Universal Robots PolyScope program: faichun_9jan_1.urp

Program faichun_9jan_1 (installation=default directory=/programs createdIn=5.11.9.1010452 lastSavedIn=5.11.9.1010452 robotSerialNumber=20225200364)
Calibrated DH parameters: a=[0.00002, -0.569483, -0.54992, -0.00001, -0.000036, 0]; d=[0.180894, -146.691669, 192.918669, -46.053088, 0.119778, 0.115602]; alpha=[1.571425, -0.001534, 0.003359, 1.568739, -1.571477, 0]; deltaTheta=[0, 0.376258, -0.101074, -0.275185, -0.000002, 0]
Robot Program (runOnlyOnce=true)
  Script file /programs/FaiChun_9 Jan_11_2.script
    | def Machining1():
    |   # Default parameters:
    |   global speed_ms = 0.05
    |   global speed_rads = 0.75
    |   global accel_mss = 3
    |   global accel_radss = 1.2
    |   global blend_radius_m = 0.0003
    | 
    |   # Add subprograms here
    |   # Start of main program
    |   # Program generated by RoboDK v5.6.8 for UR10e on 14/01/2025 11:38:46
    |   # Using nominal kinematics.
    |   blend_radius_m = 0.0003
    |   speed_ms = 0.05
    |   # set_reference(p[0.340000, -0.055000, 0.001500, 0.000000, 0.000000, 0.000000])
    |   set_tcp(p[0.000000, 0.000000, 0.252000, 0.000000, 0.000000, 0.000000])
    |   # Show Tool
    |   movej([0.533483, -1.384929, -2.455828, -0.871632, 1.570796, 2.104279],accel_radss,speed_rads,0,blend_radius_m)
    |   movel([0.533483, -1.438119, -2.486082, -0.788188, 1.570796, 2.104279],accel_mss,speed_ms,0,blend_radius_m)
    |   #SetTool1
    |   #M_RunCode6
    |   #SetRPM60000
    |   speed_ms = 0.05
    |   #M_RunCode3
    |   movel([0.533483, -1.461338, -2.497320, -0.753730, 1.570796, 2.104279],accel_mss,speed_ms,0,blend_radius_m)
    |   speed_ms = 0.003
    |   movel([0.533483, -1.467339, -2.500058, -0.744992, 1.570796, 2.104279],accel_mss,speed_ms,0,blend_radius_m)
    |   speed_ms = 0.02
    |   movel([0.259918, -1.461630, -2.504809, -0.745950, 1.570796, 1.830715],accel_mss,speed_ms,0,blend_radius_m)
    |   movel([0.369740, -1.126670, -2.705271, -0.880448, 1.570796, 1.940536],accel_mss,speed_ms,0,blend_radius_m)
    |   movel([0.742885, -1.140080, -2.699787, -0.872522, 1.570796, 2.313681],accel_mss,speed_ms,0,blend_radius_m)
    |   movel([0.533483, -1.467339, -2.500058, -0.744992, 1.570796, 2.104279],accel_mss,speed_ms,0,blend_radius_m)
    |   speed_ms = 0.003
    |   movel([0.533483, -1.461338, -2.497320, -0.753730, 1.570796, 2.104279],accel_mss,speed_ms,0,blend_radius_m)
    |   speed_ms = 0.05
    |   movel([0.533483, -1.438119, -2.486082, -0.788188, 1.570796, 2.104279],accel_mss,speed_ms,0,blend_radius_m)
    |   #M_RunCode9
    |   movel([0.533312, -1.429268, -2.493105, -0.790016, 1.570796, 2.104108],accel_mss,speed_ms,0,blend_radius_m)
    |   #M_RunCode3
    |   movel([0.533312, -1.452668, -2.504450, -0.755271, 1.570796, 2.104108],accel_mss,speed_ms,0,blend_radius_m)
    |   speed_ms = 0.003
    |   movel([0.533312, -1.458718, -2.507214, -0.746458, 1.570796, 2.104108],accel_mss,speed_ms,0,blend_radius_m)
    |   speed_ms = 0.012
    |   movel([0.529447, -1.458110, -2.507714, -0.746565, 1.570796, 2.100243],accel_mss,speed_ms,0,blend_radius_m)
    |   movel([0.527191, -1.462019, -2.504487, -0.745883, 1.570796, 2.097987],accel_mss,speed_ms,0,blend_radius_m)
    |   movel([0.521465, -1.461157, -2.505201, -0.746031, 1.570796, 2.092261],accel_mss,speed_ms,0,blend_radius_m)
    |   movel([0.523700, -1.457237, -2.508431, -0.746721, 1.570796, 2.094496],accel_mss,speed_ms,0,blend_radius_m)
    |   movel([0.521680, -1.456940, -2.508675, -0.746774, 1.570796, 2.092476],accel_mss,speed_ms,0,blend_radius_m)
    |   movel([0.519450, -1.460862, -2.505444, -0.746082, 1.570796, 2.090246],accel_mss,speed_ms,0,blend_radius_m)
    |   movel([0.514625, -1.460178, -2.506009, -0.746201, 1.570796, 2.085422],accel_mss,speed_ms,0,blend_radius_m)
    |   movel([0.513688, -1.460046, -2.506118, -0.746224, 1.570796, 2.084485],accel_mss,speed_ms,0,blend_radius_m)
    |   movel([0.516966, -1.454221, -2.510901, -0.747267, 1.570796, 2.087762],accel_mss,speed_ms,0,blend_radius_m)
    |   movel([0.520880, -1.454777, -2.510447, -0.747166, 1.570796, 2.091676],accel_mss,speed_ms,0,blend_radius_m)
    |   movel([0.522047, -1.452724, -2.512121, -0.747544, 1.570796, 2.092844],accel_mss,speed_ms,0,blend_radius_m)
    |   movel([0.516087, -1.451882, -2.512806, -0.747701, 1.570796, 2.086883],accel_mss,speed_ms,0,blend_radius_m)
    |   movel([0.511663, -1.459770, -2.506346, -0.746273, 1.570796, 2.082459],accel_mss,speed_ms,0,blend_radius_m)
    |   movel([0.510722, -1.459645, -2.506450, -0.746294, 1.570796, 2.081518],accel_mss,speed_ms,0,blend_radius_m)
    |   speed_ms = 0.02
    |   movel([0.402251, -1.451333, -2.513252, -0.747803, 1.570796, 1.973047],accel_mss,speed_ms,0,blend_radius_m)
    |   movel([0.287164, -1.455120, -2.510166, -0.747103, 1.570796, 1.857961],accel_mss,speed_ms,0,blend_radius_m)
    |   speed_ms = 0.012
    |   movel([0.289732, -1.447134, -2.516649, -0.748606, 1.570796, 1.860528],accel_mss,speed_ms,0,blend_radius_m)
    |   movel([0.283110, -1.447719, -2.516177, -0.748493, 1.570796, 1.853907],accel_mss,speed_ms,0,blend_radius_m)
    |   movel([0.282451, -1.449796, -2.514499, -0.748094, 1.570796, 1.853247],accel_mss,speed_ms,0,blend_radius_m)
    |   movel([0.286803, -1.449409, -2.514812, -0.748168, 1.570796, 1.857599],accel_mss,speed_ms,0,blend_radius_m)
    |   movel([0.284916, -1.455306, -2.510014, -0.747069, 1.570796, 1.855712],accel_mss,speed_ms,0,blend_radius_m)
    |   movel([0.283876, -1.455397, -2.509940, -0.747053, 1.570796, 1.854673],accel_mss,speed_ms,0,blend_radius_m)
    |   movel([0.278513, -1.455877, -2.509546, -0.746965, 1.570796, 1.849310],accel_mss,speed_ms,0,blend_radius_m)
    |   movel([0.279756, -1.451908, -2.512785, -0.747696, 1.570796, 1.850552],accel_mss,speed_ms,0,blend_radius_m)
    |   movel([0.277501, -1.452116, -2.512616, -0.747657, 1.570796, 1.848297],accel_mss,speed_ms,0,blend_radius_m)
    |   movel([0.276268, -1.456086, -2.509375, -0.746928, 1.570796, 1.847065],accel_mss,speed_ms,0,blend_radius_m)
    |   movel([0.269859, -1.456703, -2.508870, -0.746817, 1.570796, 1.840655],accel_mss,speed_ms,0,blend_radius_m)
    |   movel([0.271062, -1.452742, -2.512107, -0.747540, 1.570796, 1.841859],accel_mss,speed_ms,0,blend_radius_m)
    |   movel([0.266709, -1.453184, -2.511747, -0.747458, 1.570796, 1.837505],accel_mss,speed_ms,0,blend_radius_m)
    |   movel([0.268482, -1.447281, -2.516530, -0.748577, 1.570796, 1.839278],accel_mss,speed_ms,0,blend_radius_m)
    |   movel([0.272863, -1.446832, -2.516892, -0.748665, 1.570796, 1.843659],accel_mss,speed_ms,0,blend_radius_m)
    |   movel([0.273500, -1.444749, -2.518566, -0.749074, 1.570796, 1.844297],accel_mss,speed_ms,0,blend_radius_m)
    |   movel([0.269110, -1.445198, -2.518206, -0.748985, 1.570796, 1.839906],accel_mss,speed_ms,0,blend_radius_m)
    |   movel([0.270618, -1.440202, -2.522197, -0.749990, 1.570796, 1.841414],accel_mss,speed_ms,0,blend_radius_m)
    |   movel([0.270916, -1.439225, -2.522974, -0.750190, 1.570796, 1.841713],accel_mss,speed_ms,0,blend_radius_m)
    |   movel([0.277462, -1.438552, -2.523507, -0.750330, 1.570796, 1.848259],accel_mss,speed_ms,0,blend_radius_m)
    |   movel([0.276210, -1.442598, -2.520288, -0.749503, 1.570796, 1.847006],accel_mss,speed_ms,0,blend_radius_m)
    |   movel([0.278494, -1.442373, -2.520467, -0.749548, 1.570796, 1.849291],accel_mss,speed_ms,0,blend_radius_m)
    |   movel([0.280415, -1.436214, -2.525356, -0.750819, 1.570796, 1.851211],accel_mss,speed_ms,0,blend_radius_m)
    |   movel([0.271556, -1.437117, -2.524643, -0.750629, 1.570796, 1.842352],accel_mss,speed_ms,0,blend_radius_m)
    |   movel([0.309866, -1.316419, -2.609463, -0.786507, 1.570796, 1.880662],accel_mss,speed_ms,0,blend_radius_m)
    |   speed_ms = 0.02
    |   movel([0.360938, -1.167682, -2.687935, -0.856771, 1.570796, 1.931735],accel_mss,speed_ms,0,blend_radius_m)
    |   movel([0.361480, -1.166168, -2.688606, -0.857615, 1.570796, 1.932276],accel_mss,speed_ms,0,blend_radius_m)
    |   speed_ms = 0.012
    |   movel([0.373333, -1.164332, -2.689415, -0.858642, 1.570796, 1.944129],accel_mss,speed_ms,0,blend_radius_m)
    |   movel([0.376888, -1.154641, -2.693631, -0.864117, 1.570796, 1.947684],accel_mss,speed_ms,0,blend_radius_m)
    |   movel([0.373789, -1.155114, -2.693427, -0.863848, 1.570796, 1.944585],accel_mss,speed_ms,0,blend_radius_m)
    |   movel([0.371457, -1.161503, -2.690656, -0.860230, 1.570796, 1.942254],accel_mss,speed_ms,0,blend_radius_m)
    |   movel([0.362659, -1.162880, -2.690053, -0.859456, 1.570796, 1.933456],accel_mss,speed_ms,0,blend_radius_m)
    |   movel([0.363202, -1.161358, -2.690719, -0.860312, 1.570796, 1.933999],accel_mss,speed_ms,0,blend_radius_m)
    |   movel([0.366035, -1.153430, -2.694151, -0.864808, 1.570796, 1.936831],accel_mss,speed_ms,0,blend_radius_m)
    |   movel([0.372034, -1.152469, -2.694563, -0.865358, 1.570796, 1.942830],accel_mss,speed_ms,0,blend_radius_m)
    |   movel([0.373252, -1.149115, -2.695992, -0.867282, 1.570796, 1.944048],accel_mss,speed_ms,0,blend_radius_m)
    |   movel([0.367233, -1.150084, -2.695580, -0.866725, 1.570796, 1.938029],accel_mss,speed_ms,0,blend_radius_m)
    |   movel([0.370700, -1.140431, -2.699641, -0.872317, 1.570796, 1.941496],accel_mss,speed_ms,0,blend_radius_m)
    |   movel([0.376777, -1.139438, -2.700053, -0.872898, 1.570796, 1.947573],accel_mss,speed_ms,0,blend_radius_m)
    |   movel([0.379196, -1.132819, -2.702778, -0.876792, 1.570796, 1.949992],accel_mss,speed_ms,0,blend_radius_m)
    |   movel([0.388243, -1.131390, -2.703361, -0.877639, 1.570796, 1.959039],accel_mss,speed_ms,0,blend_radius_m)
    |   movel([0.385765, -1.138032, -2.700635, -0.873721, 1.570796, 1.956561],accel_mss,speed_ms,0,blend_radius_m)
    |   movel([0.388910, -1.137558, -2.700831, -0.873999, 1.570796, 1.959706],accel_mss,speed_ms,0,blend_radius_m)
    |   movel([0.391408, -1.130908, -2.703557, -0.877924, 1.570796, 1.962205],accel_mss,speed_ms,0,blend_radius_m)
    |   movel([0.400429, -1.129586, -2.704093, -0.878710, 1.570796, 1.971225],accel_mss,speed_ms,0,blend_radius_m)
    |   movel([0.396655, -1.139442, -2.700052, -0.872896, 1.570796, 1.967451],accel_mss,speed_ms,0,blend_radius_m)
    |   movel([0.390623, -1.140304, -2.699694, -0.872391, 1.570796, 1.961419],accel_mss,speed_ms,0,blend_radius_m)
    |   movel([0.389336, -1.143717, -2.698269, -0.870403, 1.570796, 1.960133],accel_mss,speed_ms,0,blend_radius_m)
    |   movel([0.398466, -1.142432, -2.698807, -0.871151, 1.570796, 1.969263],accel_mss,speed_ms,0,blend_radius_m)
    |   movel([0.403585, -1.129142, -2.704273, -0.878974, 1.570796, 1.974381],accel_mss,speed_ms,0,blend_radius_m)
    |   movel([0.563013, -1.120295, -2.707818, -0.884277, 1.570796, 2.133810],accel_mss,speed_ms,0,blend_radius_m)
    |   speed_ms = 0.02
    |   movel([0.707055, -1.139837, -2.699888, -0.872664, 1.570796, 2.277852],accel_mss,speed_ms,0,blend_radius_m)
    |   movel([0.698676, -1.152794, -2.694424, -0.865172, 1.570796, 2.269473],accel_mss,speed_ms,0,blend_radius_m)
    |   speed_ms = 0.012
    |   movel([0.706130, -1.154616, -2.693642, -0.864132, 1.570796, 2.276927],accel_mss,speed_ms,0,blend_radius_m)
    |   movel([0.708299, -1.151299, -2.695063, -0.866028, 1.570796, 2.279096],accel_mss,speed_ms,0,blend_radius_m)
    |   movel([0.703392, -1.150081, -2.695581, -0.866727, 1.570796, 2.274188],accel_mss,speed_ms,0,blend_radius_m)
    |   movel([0.709631, -1.140484, -2.699619, -0.872286, 1.570796, 2.280428],accel_mss,speed_ms,0,blend_radius_m)
    |   movel([0.710822, -1.140781, -2.699495, -0.872113, 1.570796, 2.281618],accel_mss,speed_ms,0,blend_radius_m)
    |   movel([0.716930, -1.142343, -2.698844, -0.871202, 1.570796, 2.287726],accel_mss,speed_ms,0,blend_radius_m)
    |   movel([0.712681, -1.148808, -2.696122, -0.867459, 1.570796, 2.283477],accel_mss,speed_ms,0,blend_radius_m)
    |   movel([0.715213, -1.149470, -2.695841, -0.867078, 1.570796, 2.286009],accel_mss,speed_ms,0,blend_radius_m)
    |   movel([0.719478, -1.143013, -2.698564, -0.870812, 1.570796, 2.290274],accel_mss,speed_ms,0,blend_radius_m)
    |   movel([0.726693, -1.144971, -2.697742, -0.869675, 1.570796, 2.297489],accel_mss,speed_ms,0,blend_radius_m)
    |   movel([0.722404, -1.151397, -2.695021, -0.865972, 1.570796, 2.293201],accel_mss,speed_ms,0,blend_radius_m)
    |   movel([0.727224, -1.152737, -2.694448, -0.865204, 1.570796, 2.298021],accel_mss,speed_ms,0,blend_radius_m)
    |   movel([0.720946, -1.162096, -2.690396, -0.859897, 1.570796, 2.291743],accel_mss,speed_ms,0,blend_radius_m)
    |   movel([0.716151, -1.160787, -2.690968, -0.860634, 1.570796, 2.286947],accel_mss,speed_ms,0,blend_radius_m)
    |   movel([0.713986, -1.164044, -2.689542, -0.858803, 1.570796, 2.284782],accel_mss,speed_ms,0,blend_radius_m)
    |   movel([0.718770, -1.165346, -2.688968, -0.858075, 1.570796, 2.289566],accel_mss,speed_ms,0,blend_radius_m)
    |   movel([0.713629, -1.173035, -2.685547, -0.853807, 1.570796, 2.284425],accel_mss,speed_ms,0,blend_radius_m)
    |   movel([0.712640, -1.174516, -2.684881, -0.852992, 1.570796, 2.283436],accel_mss,speed_ms,0,blend_radius_m)
    |   movel([0.705579, -1.172648, -2.685720, -0.854020, 1.570796, 2.276375],accel_mss,speed_ms,0,blend_radius_m)
    |   movel([0.709681, -1.166442, -2.688485, -0.857463, 1.570796, 2.280478],accel_mss,speed_ms,0,blend_radius_m)
    |   movel([0.707181, -1.165792, -2.688772, -0.857825, 1.570796, 2.277978],accel_mss,speed_ms,0,blend_radius_m)
    |   movel([0.700980, -1.175214, -2.684566, -0.852609, 1.570796, 2.271776],accel_mss,speed_ms,0,blend_radius_m)
    |   movel([0.710514, -1.177702, -2.683440, -0.851247, 1.570796, 2.281311],accel_mss,speed_ms,0,blend_radius_m)
    |   speed_ms = 0.02
    |   movel([0.615153, -1.324265, -2.604567, -0.783557, 1.570796, 2.185950],accel_mss,speed_ms,0,blend_radius_m)
    |   movel([0.542601, -1.442874, -2.520067, -0.749448, 1.570796, 2.113397],accel_mss,speed_ms,0,blend_radius_m)
    |   speed_ms = 0.012
    |   movel([0.534737, -1.441630, -2.521060, -0.749699, 1.570796, 2.105533],accel_mss,speed_ms,0,blend_radius_m)
    |   movel([0.531216, -1.447708, -2.516186, -0.748495, 1.570796, 2.102013],accel_mss,speed_ms,0,blend_radius_m)
    |   movel([0.533250, -1.448021, -2.515933, -0.748434, 1.570796, 2.104046],accel_mss,speed_ms,0,blend_radius_m)
    |   movel([0.535568, -1.444031, -2.519142, -0.749216, 1.570796, 2.106364],accel_mss,speed_ms,0,blend_radius_m)
    |   movel([0.541367, -1.444954, -2.518401, -0.749033, 1.570796, 2.112164],accel_mss,speed_ms,0,blend_radius_m)
    |   movel([0.540803, -1.445915, -2.517630, -0.748844, 1.570796, 2.111599],accel_mss,speed_ms,0,blend_radius_m)
    |   movel([0.537910, -1.450844, -2.513649, -0.747896, 1.570796, 2.108707],accel_mss,speed_ms,0,blend_radius_m)
    |   movel([0.534018, -1.450225, -2.514152, -0.748013, 1.570796, 2.104814],accel_mss,speed_ms,0,blend_radius_m)
    |   movel([0.532824, -1.452279, -2.512483, -0.747626, 1.570796, 2.103621],accel_mss,speed_ms,0,blend_radius_m)
    |   movel([0.536712, -1.452896, -2.511981, -0.747512, 1.570796, 2.107508],accel_mss,speed_ms,0,blend_radius_m)
    |   movel([0.533312, -1.458718, -2.507214, -0.746458, 1.570796, 2.104108],accel_mss,speed_ms,0,blend_radius_m)
    |   speed_ms = 0.003
    |   movel([0.533312, -1.452668, -2.504450, -0.755271, 1.570796, 2.104108],accel_mss,speed_ms,0,blend_radius_m)
    |   speed_ms = 0.05
    |   movel([0.533312, -1.429268, -2.493105, -0.790016, 1.570796, 2.104108],accel_mss,speed_ms,0,blend_radius_m)
    |   #M_RunCode9
    |   movel([0.417526, -1.170993, -2.652148, -0.889248, 1.570796, 1.988323],accel_mss,speed_ms,0,blend_radius_m)
    |   #M_RunCode3
    |   # num 0 inside
    |   movel([0.417526, -1.198293, -2.666816, -0.847281, 1.570796, 1.988323],accel_mss,speed_ms,0,blend_radius_m)
    |   speed_ms = 0.003
    |   movel([0.417526, -1.205477, -2.670419, -0.836494, 1.570796, 1.988323],accel_mss,speed_ms,0,blend_radius_m)
    |   speed_ms = 0.015
    |   movel([0.408855, -1.212168, -2.667155, -0.833065, 1.570796, 1.979651],accel_mss,speed_ms,0,blend_radius_m)
    |   movel([0.402561, -1.216461, -2.665035, -0.830893, 1.570796, 1.973358],accel_mss,speed_ms,0,blend_radius_m)
    |   movel([0.400243, -1.217697, -2.664421, -0.830271, 1.570796, 1.971039],accel_mss,speed_ms,0,blend_radius_m)
    |   movel([0.398416, -1.218288, -2.664127, -0.829974, 1.570796, 1.969213],accel_mss,speed_ms,0,blend_radius_m)
    |   movel([0.397079, -1.218242, -2.664149, -0.829997, 1.570796, 1.967875],accel_mss,speed_ms,0,blend_radius_m)
    |   movel([0.396226, -1.217555, -2.664492, -0.830342, 1.570796, 1.967022],accel_mss,speed_ms,0,blend_radius_m)
    |   movel([0.395959, -1.216391, -2.665070, -0.830928, 1.570796, 1.966756],accel_mss,speed_ms,0,blend_radius_m)
    |   movel([0.396382, -1.214913, -2.665802, -0.831674, 1.570796, 1.967179],accel_mss,speed_ms,0,blend_radius_m)
    |   movel([0.397498, -1.213118, -2.666688, -0.832583, 1.570796, 1.968295],accel_mss,speed_ms,0,blend_radius_m)
    |   movel([0.399310, -1.211002, -2.667728, -0.833659, 1.570796, 1.970106],accel_mss,speed_ms,0,blend_radius_m)
    |   movel([0.405022, -1.205584, -2.670367, -0.836438, 1.570796, 1.975818],accel_mss,speed_ms,0,blend_radius_m)
    |   movel([0.413543, -1.198419, -2.673807, -0.840163, 1.570796, 1.984339],accel_mss,speed_ms,0,blend_radius_m)
    |   movel([0.422369, -1.191559, -2.677048, -0.843782, 1.570796, 1.993165],accel_mss,speed_ms,0,blend_radius_m)
    |   movel([0.428878, -1.187122, -2.679117, -0.846150, 1.570796, 1.999674],accel_mss,speed_ms,0,blend_radius_m)
    |   movel([0.431283, -1.185853, -2.679705, -0.846831, 1.570796, 2.002079],accel_mss,speed_ms,0,blend_radius_m)
    |   movel([0.433167, -1.185257, -2.679980, -0.847152, 1.570796, 2.003963],accel_mss,speed_ms,0,blend_radius_m)
    |   movel([0.434527, -1.185338, -2.679943, -0.847108, 1.570796, 2.005323],accel_mss,speed_ms,0,blend_radius_m)
    |   movel([0.435362, -1.186094, -2.679593, -0.846702, 1.570796, 2.006158],accel_mss,speed_ms,0,blend_radius_m)
    |   movel([0.435577, -1.187342, -2.679015, -0.846032, 1.570796, 2.006373],accel_mss,speed_ms,0,blend_radius_m)
    |   movel([0.435084, -1.188898, -2.678291, -0.845200, 1.570796, 2.005880],accel_mss,speed_ms,0,blend_radius_m)
    |   movel([0.433878, -1.190761, -2.677421, -0.844206, 1.570796, 2.004675],accel_mss,speed_ms,0,blend_radius_m)
    |   movel([0.431974, -1.192924, -2.676407, -0.843058, 1.570796, 2.002770],accel_mss,speed_ms,0,blend_radius_m)
    |   movel([0.426094, -1.198383, -2.673824, -0.840182, 1.570796, 1.996890],accel_mss,speed_ms,0,blend_radius_m)
    |   movel([0.417526, -1.205477, -2.670419, -0.836494, 1.570796, 1.988323],accel_mss,speed_ms,0,blend_radius_m)
    |   speed_ms = 0.003
    |   movel([0.417526, -1.198293, -2.666816, -0.847281, 1.570796, 1.988323],accel_mss,speed_ms,0,blend_radius_m)
    |   speed_ms = 0.05
    |   movel([0.417526, -1.170993, -2.652148, -0.889248, 1.570796, 1.988323],accel_mss,speed_ms,0,blend_radius_m)
    |   #M_RunCode9
    |   movel([0.421749, -1.178679, -2.648562, -0.885148, 1.570796, 1.992545],accel_mss,speed_ms,0,blend_radius_m)
    |   #M_RunCode3
    |   #num 0 outside
    |   movel([0.421749, -1.205919, -2.663128, -0.843342, 1.570796, 1.992545],accel_mss,speed_ms,0,blend_radius_m)
    |   speed_ms = 0.003
    |   movel([0.421749, -1.213083, -2.666705, -0.832601, 1.570796, 1.992545],accel_mss,speed_ms,0,blend_radius_m)
    |   speed_ms = 0.015
    |   movel([0.418589, -1.215448, -2.665537, -0.831403, 1.570796, 1.989385],accel_mss,speed_ms,0,blend_radius_m)
    |   movel([0.415567, -1.217446, -2.664546, -0.830397, 1.570796, 1.986363],accel_mss,speed_ms,0,blend_radius_m)
    |   movel([0.412674, -1.219085, -2.663729, -0.829575, 1.570796, 1.983470],accel_mss,speed_ms,0,blend_radius_m)
    |   movel([0.409911, -1.220363, -2.663090, -0.828936, 1.570796, 1.980707],accel_mss,speed_ms,0,blend_radius_m)
    |   movel([0.407315, -1.221290, -2.662626, -0.828474, 1.570796, 1.978111],accel_mss,speed_ms,0,blend_radius_m)
    |   movel([0.404924, -1.221871, -2.662334, -0.828184, 1.570796, 1.975720],accel_mss,speed_ms,0,blend_radius_m)
    |   movel([0.402734, -1.222111, -2.662214, -0.828065, 1.570796, 1.973530],accel_mss,speed_ms,0,blend_radius_m)
    |   movel([0.400748, -1.222003, -2.662268, -0.828118, 1.570796, 1.971545],accel_mss,speed_ms,0,blend_radius_m)
    |   movel([0.398984, -1.221568, -2.662486, -0.828335, 1.570796, 1.969780],accel_mss,speed_ms,0,blend_radius_m)
    |   movel([0.397463, -1.220832, -2.662856, -0.828702, 1.570796, 1.968260],accel_mss,speed_ms,0,blend_radius_m)
    |   movel([0.396184, -1.219786, -2.663379, -0.829224, 1.570796, 1.966980],accel_mss,speed_ms,0,blend_radius_m)
    |   movel([0.395146, -1.218434, -2.664054, -0.829901, 1.570796, 1.965942],accel_mss,speed_ms,0,blend_radius_m)
    |   movel([0.394396, -1.216841, -2.664847, -0.830701, 1.570796, 1.965192],accel_mss,speed_ms,0,blend_radius_m)
    |   movel([0.393982, -1.215084, -2.665718, -0.831587, 1.570796, 1.964778],accel_mss,speed_ms,0,blend_radius_m)
    |   movel([0.393900, -1.213162, -2.666666, -0.832561, 1.570796, 1.964697],accel_mss,speed_ms,0,blend_radius_m)
    |   movel([0.394161, -1.211065, -2.667697, -0.833627, 1.570796, 1.964958],accel_mss,speed_ms,0,blend_radius_m)
    |   movel([0.394772, -1.208828, -2.668790, -0.834770, 1.570796, 1.965568],accel_mss,speed_ms,0,blend_radius_m)
    |   movel([0.395745, -1.206481, -2.669932, -0.835976, 1.570796, 1.966541],accel_mss,speed_ms,0,blend_radius_m)
    |   movel([0.397083, -1.204017, -2.671124, -0.837248, 1.570796, 1.967879],accel_mss,speed_ms,0,blend_radius_m)
    |   movel([0.398791, -1.201439, -2.672364, -0.838586, 1.570796, 1.969588],accel_mss,speed_ms,0,blend_radius_m)
    |   movel([0.400858, -1.198792, -2.673629, -0.839968, 1.570796, 1.971654],accel_mss,speed_ms,0,blend_radius_m)
    |   movel([0.403274, -1.196129, -2.674894, -0.841365, 1.570796, 1.974071],accel_mss,speed_ms,0,blend_radius_m)
    |   movel([0.406040, -1.193452, -2.676159, -0.842778, 1.570796, 1.976836],accel_mss,speed_ms,0,blend_radius_m)
    |   movel([0.409156, -1.190762, -2.677421, -0.844206, 1.570796, 1.979952],accel_mss,speed_ms,0,blend_radius_m)
    |   movel([0.412397, -1.188248, -2.678594, -0.845547, 1.570796, 1.983193],accel_mss,speed_ms,0,blend_radius_m)
    |   movel([0.415520, -1.186109, -2.679587, -0.846694, 1.570796, 1.986317],accel_mss,speed_ms,0,blend_radius_m)
    |   movel([0.418526, -1.184345, -2.680401, -0.847643, 1.570796, 1.989323],accel_mss,speed_ms,0,blend_radius_m)
    |   movel([0.421407, -1.182966, -2.681036, -0.848387, 1.570796, 1.992203],accel_mss,speed_ms,0,blend_radius_m)
    |   movel([0.424115, -1.181967, -2.681494, -0.848928, 1.570796, 1.994911],accel_mss,speed_ms,0,blend_radius_m)
    |   movel([0.426598, -1.181352, -2.681776, -0.849261, 1.570796, 1.997394],accel_mss,speed_ms,0,blend_radius_m)
    |   movel([0.428858, -1.181116, -2.681884, -0.849389, 1.570796, 1.999654],accel_mss,speed_ms,0,blend_radius_m)
    |   movel([0.430890, -1.181265, -2.681816, -0.849308, 1.570796, 2.001686],accel_mss,speed_ms,0,blend_radius_m)
    |   movel([0.432671, -1.181770, -2.681585, -0.849034, 1.570796, 2.003468],accel_mss,speed_ms,0,blend_radius_m)
    |   movel([0.434190, -1.182603, -2.681203, -0.848584, 1.570796, 2.004986],accel_mss,speed_ms,0,blend_radius_m)
    |   movel([0.435445, -1.183761, -2.680670, -0.847958, 1.570796, 2.006242],accel_mss,speed_ms,0,blend_radius_m)
    |   movel([0.436432, -1.185242, -2.679987, -0.847160, 1.570796, 2.007229],accel_mss,speed_ms,0,blend_radius_m)
    |   movel([0.437113, -1.186965, -2.679190, -0.846234, 1.570796, 2.007909],accel_mss,speed_ms,0,blend_radius_m)
    |   movel([0.437449, -1.188842, -2.678317, -0.845230, 1.570796, 2.008245],accel_mss,speed_ms,0,blend_radius_m)
    |   movel([0.437439, -1.190873, -2.677369, -0.844147, 1.570796, 2.008236],accel_mss,speed_ms,0,blend_radius_m)
    |   movel([0.437088, -1.193056, -2.676345, -0.842988, 1.570796, 2.007885],accel_mss,speed_ms,0,blend_radius_m)
    |   movel([0.436387, -1.195356, -2.675260, -0.841773, 1.570796, 2.007183],accel_mss,speed_ms,0,blend_radius_m)
    |   movel([0.435324, -1.197746, -2.674127, -0.840516, 1.570796, 2.006120],accel_mss,speed_ms,0,blend_radius_m)
    |   movel([0.433899, -1.200225, -2.672945, -0.839219, 1.570796, 2.004695],accel_mss,speed_ms,0,blend_radius_m)
    |   movel([0.432120, -1.202788, -2.671716, -0.837885, 1.570796, 2.002916],accel_mss,speed_ms,0,blend_radius_m)
    |   movel([0.430005, -1.205384, -2.670464, -0.836542, 1.570796, 2.000801],accel_mss,speed_ms,0,blend_radius_m)
    |   movel([0.427569, -1.207965, -2.669211, -0.835213, 1.570796, 1.998365],accel_mss,speed_ms,0,blend_radius_m)
    |   movel([0.424816, -1.210531, -2.667958, -0.833900, 1.570796, 1.995612],accel_mss,speed_ms,0,blend_radius_m)
    |   movel([0.421749, -1.213083, -2.666705, -0.832601, 1.570796, 1.992545],accel_mss,speed_ms,0,blend_radius_m)
    |   speed_ms = 0.003
    |   movel([0.421749, -1.205919, -2.663128, -0.843342, 1.570796, 1.992545],accel_mss,speed_ms,0,blend_radius_m)
    |   speed_ms = 0.05
    |   movel([0.421749, -1.178679, -2.648562, -0.885148, 1.570796, 1.992545],accel_mss,speed_ms,0,blend_radius_m)
    |   #M_RunCode9
    |   movel([0.398548, -1.160673, -2.656867, -0.894849, 1.570796, 1.969344],accel_mss,speed_ms,0,blend_radius_m)
    |   #M_RunCode3
    |   # num 2
    |   movel([0.398548, -1.188046, -2.671670, -0.852673, 1.570796, 1.969344],accel_mss,speed_ms,0,blend_radius_m)
    |   speed_ms = 0.003
    |   movel([0.398548, -1.195256, -2.675308, -0.841825, 1.570796, 1.969344],accel_mss,speed_ms,0,blend_radius_m)
    |   speed_ms = 0.02
    |   movel([0.387519, -1.204390, -2.670944, -0.837055, 1.570796, 1.958316],accel_mss,speed_ms,0,blend_radius_m)
    |   movel([0.373276, -1.182200, -2.681388, -0.848802, 1.570796, 1.944072],accel_mss,speed_ms,0,blend_radius_m)
    |   movel([0.374391, -1.181239, -2.681828, -0.849322, 1.570796, 1.945187],accel_mss,speed_ms,0,blend_radius_m)
    |   movel([0.377402, -1.179045, -2.682829, -0.850514, 1.570796, 1.948199],accel_mss,speed_ms,0,blend_radius_m)
    |   movel([0.380700, -1.177412, -2.683572, -0.851406, 1.570796, 1.951496],accel_mss,speed_ms,0,blend_radius_m)
    |   movel([0.384107, -1.176260, -2.684093, -0.852036, 1.570796, 1.954903],accel_mss,speed_ms,0,blend_radius_m)
    |   movel([0.387437, -1.175507, -2.684433, -0.852448, 1.570796, 1.958233],accel_mss,speed_ms,0,blend_radius_m)
    |   movel([0.396101, -1.174407, -2.684930, -0.853052, 1.570796, 1.966897],accel_mss,speed_ms,0,blend_radius_m)
    |   movel([0.404086, -1.173536, -2.685322, -0.853531, 1.570796, 1.974882],accel_mss,speed_ms,0,blend_radius_m)
    |   movel([0.407182, -1.172914, -2.685601, -0.853874, 1.570796, 1.977978],accel_mss,speed_ms,0,blend_radius_m)
    |   movel([0.410285, -1.171948, -2.686034, -0.854407, 1.570796, 1.981082],accel_mss,speed_ms,0,blend_radius_m)
    |   movel([0.413245, -1.170575, -2.686648, -0.855166, 1.570796, 1.984041],accel_mss,speed_ms,0,blend_radius_m)
    |   movel([0.415914, -1.168726, -2.687472, -0.856191, 1.570796, 1.986710],accel_mss,speed_ms,0,blend_radius_m)
    |   movel([0.418722, -1.165926, -2.688712, -0.857750, 1.570796, 1.989518],accel_mss,speed_ms,0,blend_radius_m)
    |   movel([0.419689, -1.164533, -2.689327, -0.858530, 1.570796, 1.990485],accel_mss,speed_ms,0,blend_radius_m)
    |   movel([0.420364, -1.163144, -2.689937, -0.859308, 1.570796, 1.991160],accel_mss,speed_ms,0,blend_radius_m)
    |   movel([0.420918, -1.160616, -2.691043, -0.860730, 1.570796, 1.991714],accel_mss,speed_ms,0,blend_radius_m)
    |   movel([0.420451, -1.158600, -2.691920, -0.861869, 1.570796, 1.991247],accel_mss,speed_ms,0,blend_radius_m)
    |   movel([0.419659, -1.157633, -2.692340, -0.862417, 1.570796, 1.990456],accel_mss,speed_ms,0,blend_radius_m)
    |   movel([0.418681, -1.157242, -2.692509, -0.862638, 1.570796, 1.989477],accel_mss,speed_ms,0,blend_radius_m)
    |   movel([0.417618, -1.157384, -2.692447, -0.862558, 1.570796, 1.988414],accel_mss,speed_ms,0,blend_radius_m)
    |   movel([0.416582, -1.158002, -2.692180, -0.862208, 1.570796, 1.987378],accel_mss,speed_ms,0,blend_radius_m)
    |   movel([0.415423, -1.159560, -2.691503, -0.861326, 1.570796, 1.986220],accel_mss,speed_ms,0,blend_radius_m)
    |   movel([0.414382, -1.161128, -2.690820, -0.860442, 1.570796, 1.985179],accel_mss,speed_ms,0,blend_radius_m)
    |   movel([0.412740, -1.162760, -2.690106, -0.859524, 1.570796, 1.983536],accel_mss,speed_ms,0,blend_radius_m)
    |   movel([0.410524, -1.164199, -2.689473, -0.858716, 1.570796, 1.981321],accel_mss,speed_ms,0,blend_radius_m)
    |   movel([0.408517, -1.164649, -2.689276, -0.858464, 1.570796, 1.979313],accel_mss,speed_ms,0,blend_radius_m)
    |   movel([0.406864, -1.164233, -2.689459, -0.858697, 1.570796, 1.977661],accel_mss,speed_ms,0,blend_radius_m)
    |   movel([0.405717, -1.163077, -2.689966, -0.859345, 1.570796, 1.976513],accel_mss,speed_ms,0,blend_radius_m)
    |   movel([0.405200, -1.161391, -2.690705, -0.860293, 1.570796, 1.975996],accel_mss,speed_ms,0,blend_radius_m)
    |   movel([0.405438, -1.159373, -2.691584, -0.861432, 1.570796, 1.976234],accel_mss,speed_ms,0,blend_radius_m)
    |   movel([0.406483, -1.157237, -2.692511, -0.862641, 1.570796, 1.977279],accel_mss,speed_ms,0,blend_radius_m)
    |   movel([0.408389, -1.155207, -2.693387, -0.863795, 1.570796, 1.979185],accel_mss,speed_ms,0,blend_radius_m)
    |   movel([0.410308, -1.153825, -2.693981, -0.864583, 1.570796, 1.981104],accel_mss,speed_ms,0,blend_radius_m)
    |   movel([0.412191, -1.152957, -2.694353, -0.865078, 1.570796, 1.982988],accel_mss,speed_ms,0,blend_radius_m)
    |   movel([0.414040, -1.152604, -2.694505, -0.865280, 1.570796, 1.984836],accel_mss,speed_ms,0,blend_radius_m)
    |   movel([0.415848, -1.152773, -2.694432, -0.865184, 1.570796, 1.986644],accel_mss,speed_ms,0,blend_radius_m)
    |   movel([0.417547, -1.153401, -2.694163, -0.864825, 1.570796, 1.988343],accel_mss,speed_ms,0,blend_radius_m)
    |   movel([0.419078, -1.154418, -2.693726, -0.864244, 1.570796, 1.989874],accel_mss,speed_ms,0,blend_radius_m)
    |   movel([0.421621, -1.157629, -2.692341, -0.862419, 1.570796, 1.992417],accel_mss,speed_ms,0,blend_radius_m)
    |   movel([0.422740, -1.160129, -2.691255, -0.861004, 1.570796, 1.993536],accel_mss,speed_ms,0,blend_radius_m)
    |   movel([0.423427, -1.162792, -2.690091, -0.859505, 1.570796, 1.994224],accel_mss,speed_ms,0,blend_radius_m)
    |   movel([0.423686, -1.165609, -2.688852, -0.857927, 1.570796, 1.994483],accel_mss,speed_ms,0,blend_radius_m)
    |   movel([0.423519, -1.168579, -2.687537, -0.856272, 1.570796, 1.994315],accel_mss,speed_ms,0,blend_radius_m)
    |   movel([0.422775, -1.171579, -2.686200, -0.854611, 1.570796, 1.993571],accel_mss,speed_ms,0,blend_radius_m)
    |   movel([0.421289, -1.174496, -2.684890, -0.853003, 1.570796, 1.992085],accel_mss,speed_ms,0,blend_radius_m)
    |   movel([0.419070, -1.177328, -2.683609, -0.851451, 1.570796, 1.989866],accel_mss,speed_ms,0,blend_radius_m)
    |   movel([0.416125, -1.180080, -2.682358, -0.849952, 1.570796, 1.986922],accel_mss,speed_ms,0,blend_radius_m)
    |   movel([0.413191, -1.182183, -2.681395, -0.848811, 1.570796, 1.983988],accel_mss,speed_ms,0,blend_radius_m)
    |   movel([0.410228, -1.183711, -2.680693, -0.847984, 1.570796, 1.981024],accel_mss,speed_ms,0,blend_radius_m)
    |   movel([0.407305, -1.184765, -2.680207, -0.847416, 1.570796, 1.978101],accel_mss,speed_ms,0,blend_radius_m)
    |   movel([0.404499, -1.185444, -2.679894, -0.847051, 1.570796, 1.975295],accel_mss,speed_ms,0,blend_radius_m)
    |   movel([0.397845, -1.186264, -2.679515, -0.846611, 1.570796, 1.968641],accel_mss,speed_ms,0,blend_radius_m)
    |   movel([0.391540, -1.187111, -2.679122, -0.846156, 1.570796, 1.962337],accel_mss,speed_ms,0,blend_radius_m)
    |   movel([0.388986, -1.187747, -2.678827, -0.845815, 1.570796, 1.959782],accel_mss,speed_ms,0,blend_radius_m)
    |   movel([0.386370, -1.188709, -2.678379, -0.845301, 1.570796, 1.957167],accel_mss,speed_ms,0,blend_radius_m)
    |   movel([0.383776, -1.190069, -2.677745, -0.844575, 1.570796, 1.954572],accel_mss,speed_ms,0,blend_radius_m)
    |   movel([0.381297, -1.191889, -2.676893, -0.843607, 1.570796, 1.952094],accel_mss,speed_ms,0,blend_radius_m)
    |   movel([0.381830, -1.192722, -2.676502, -0.843165, 1.570796, 1.952626],accel_mss,speed_ms,0,blend_radius_m)
    |   movel([0.383468, -1.194889, -2.675481, -0.842019, 1.570796, 1.954264],accel_mss,speed_ms,0,blend_radius_m)
    |   movel([0.385262, -1.196485, -2.674726, -0.841178, 1.570796, 1.956059],accel_mss,speed_ms,0,blend_radius_m)
    |   movel([0.387208, -1.197517, -2.674236, -0.840636, 1.570796, 1.958005],accel_mss,speed_ms,0,blend_radius_m)
    |   movel([0.389316, -1.197985, -2.674013, -0.840391, 1.570796, 1.960112],accel_mss,speed_ms,0,blend_radius_m)
    |   movel([0.391528, -1.197956, -2.674027, -0.840406, 1.570796, 1.962325],accel_mss,speed_ms,0,blend_radius_m)
    |   movel([0.393803, -1.197493, -2.674247, -0.840649, 1.570796, 1.964599],accel_mss,speed_ms,0,blend_radius_m)
    |   movel([0.396140, -1.196594, -2.674674, -0.841121, 1.570796, 1.966936],accel_mss,speed_ms,0,blend_radius_m)
    |   movel([0.398548, -1.195256, -2.675308, -0.841825, 1.570796, 1.969344],accel_mss,speed_ms,0,blend_radius_m)
    |   speed_ms = 0.003
    |   movel([0.398548, -1.188046, -2.671670, -0.852673, 1.570796, 1.969344],accel_mss,speed_ms,0,blend_radius_m)
    |   speed_ms = 0.05
    |   movel([0.398548, -1.160673, -2.656867, -0.894849, 1.570796, 1.969344],accel_mss,speed_ms,0,blend_radius_m)
    |   #M_RunCode9
    |   movel([0.492183, -1.374535, -2.534046, -0.803807, 1.570796, 2.062980],accel_mss,speed_ms,0,blend_radius_m)
    |   #M_RunCode3
    |   movel([0.492183, -1.399008, -2.546063, -0.767317, 1.570796, 2.062980],accel_mss,speed_ms,0,blend_radius_m)
    |   speed_ms = 0.003
    |   movel([0.492183, -1.405355, -2.548996, -0.758039, 1.570796, 2.062980],accel_mss,speed_ms,0,blend_radius_m)
    |   speed_ms = 0.02
    |   movel([0.494554, -1.404214, -2.549842, -0.758333, 1.570796, 2.065351],accel_mss,speed_ms,0,blend_radius_m)
    |   movel([0.497069, -1.403547, -2.550337, -0.758505, 1.570796, 2.067866],accel_mss,speed_ms,0,blend_radius_m)
    |   movel([0.499611, -1.403261, -2.550549, -0.758580, 1.570796, 2.070408],accel_mss,speed_ms,0,blend_radius_m)
    |   movel([0.502055, -1.403267, -2.550544, -0.758578, 1.570796, 2.072851],accel_mss,speed_ms,0,blend_radius_m)
    |   movel([0.508325, -1.403916, -2.550063, -0.758410, 1.570796, 2.079121],accel_mss,speed_ms,0,blend_radius_m)
    |   movel([0.514086, -1.404611, -2.549548, -0.758230, 1.570796, 2.084883],accel_mss,speed_ms,0,blend_radius_m)
    |   movel([0.516344, -1.404668, -2.549506, -0.758215, 1.570796, 2.087141],accel_mss,speed_ms,0,blend_radius_m)
    |   movel([0.518640, -1.404466, -2.549656, -0.758268, 1.570796, 2.089437],accel_mss,speed_ms,0,blend_radius_m)
    |   movel([0.520871, -1.403935, -2.550049, -0.758405, 1.570796, 2.091667],accel_mss,speed_ms,0,blend_radius_m)
    |   movel([0.522937, -1.403002, -2.550740, -0.758647, 1.570796, 2.093733],accel_mss,speed_ms,0,blend_radius_m)
    |   movel([0.525186, -1.401385, -2.551934, -0.759070, 1.570796, 2.095982],accel_mss,speed_ms,0,blend_radius_m)
    |   movel([0.525999, -1.400510, -2.552579, -0.759300, 1.570796, 2.096795],accel_mss,speed_ms,0,blend_radius_m)
    |   movel([0.526604, -1.399591, -2.553255, -0.759543, 1.570796, 2.097401],accel_mss,speed_ms,0,blend_radius_m)
    |   movel([0.527228, -1.397806, -2.554564, -0.760019, 1.570796, 2.098024],accel_mss,speed_ms,0,blend_radius_m)
    |   movel([0.527082, -1.396230, -2.555715, -0.760443, 1.570796, 2.097878],accel_mss,speed_ms,0,blend_radius_m)
    |   movel([0.526613, -1.395377, -2.556338, -0.760674, 1.570796, 2.097409],accel_mss,speed_ms,0,blend_radius_m)
    |   movel([0.525954, -1.394923, -2.556668, -0.760798, 1.570796, 2.096751],accel_mss,speed_ms,0,blend_radius_m)
    |   movel([0.525193, -1.394847, -2.556724, -0.760818, 1.570796, 2.095990],accel_mss,speed_ms,0,blend_radius_m)
    |   movel([0.524404, -1.395130, -2.556518, -0.760741, 1.570796, 2.095201],accel_mss,speed_ms,0,blend_radius_m)
    |   movel([0.523441, -1.396092, -2.555816, -0.760481, 1.570796, 2.094237],accel_mss,speed_ms,0,blend_radius_m)
    |   movel([0.522557, -1.397084, -2.555092, -0.760213, 1.570796, 2.093354],accel_mss,speed_ms,0,blend_radius_m)
    |   movel([0.521242, -1.398019, -2.554408, -0.759962, 1.570796, 2.092038],accel_mss,speed_ms,0,blend_radius_m)
    |   movel([0.519539, -1.398719, -2.553894, -0.759775, 1.570796, 2.090335],accel_mss,speed_ms,0,blend_radius_m)
    |   movel([0.518076, -1.398712, -2.553900, -0.759777, 1.570796, 2.088872],accel_mss,speed_ms,0,blend_radius_m)
    |   movel([0.516943, -1.398121, -2.554333, -0.759935, 1.570796, 2.087739],accel_mss,speed_ms,0,blend_radius_m)
    |   movel([0.516241, -1.397065, -2.555106, -0.760218, 1.570796, 2.087037],accel_mss,speed_ms,0,blend_radius_m)
    |   movel([0.516038, -1.395715, -2.556091, -0.760583, 1.570796, 2.086834],accel_mss,speed_ms,0,blend_radius_m)
    |   movel([0.516399, -1.394250, -2.557158, -0.760981, 1.570796, 2.087195],accel_mss,speed_ms,0,blend_radius_m)
    |   movel([0.517341, -1.392838, -2.558183, -0.761368, 1.570796, 2.088137],accel_mss,speed_ms,0,blend_radius_m)
    |   movel([0.518880, -1.391654, -2.559040, -0.761695, 1.570796, 2.089676],accel_mss,speed_ms,0,blend_radius_m)
    |   movel([0.520364, -1.390953, -2.559547, -0.761889, 1.570796, 2.091161],accel_mss,speed_ms,0,blend_radius_m)
    |   movel([0.521777, -1.390632, -2.559779, -0.761979, 1.570796, 2.092573],accel_mss,speed_ms,0,blend_radius_m)
    |   movel([0.523112, -1.390689, -2.559738, -0.761963, 1.570796, 2.093908],accel_mss,speed_ms,0,blend_radius_m)
    |   movel([0.524369, -1.391124, -2.559423, -0.761842, 1.570796, 2.095165],accel_mss,speed_ms,0,blend_radius_m)
    |   movel([0.525510, -1.391878, -2.558878, -0.761633, 1.570796, 2.096306],accel_mss,speed_ms,0,blend_radius_m)
    |   movel([0.526495, -1.392895, -2.558141, -0.761352, 1.570796, 2.097291],accel_mss,speed_ms,0,blend_radius_m)
    |   movel([0.527999, -1.395705, -2.556099, -0.760585, 1.570796, 2.098795],accel_mss,speed_ms,0,blend_radius_m)
    |   movel([0.528561, -1.397751, -2.554604, -0.760034, 1.570796, 2.099357],accel_mss,speed_ms,0,blend_radius_m)
    |   movel([0.528805, -1.399842, -2.553070, -0.759477, 1.570796, 2.099602],accel_mss,speed_ms,0,blend_radius_m)
    |   movel([0.528733, -1.401977, -2.551497, -0.758914, 1.570796, 2.099529],accel_mss,speed_ms,0,blend_radius_m)
    |   movel([0.528346, -1.404157, -2.549884, -0.758347, 1.570796, 2.099142],accel_mss,speed_ms,0,blend_radius_m)
    |   movel([0.527544, -1.406266, -2.548318, -0.757805, 1.570796, 2.098340],accel_mss,speed_ms,0,blend_radius_m)
    |   movel([0.526223, -1.408195, -2.546879, -0.757315, 1.570796, 2.097019],accel_mss,speed_ms,0,blend_radius_m)
    |   movel([0.524388, -1.409944, -2.545570, -0.756875, 1.570796, 2.095185],accel_mss,speed_ms,0,blend_radius_m)
    |   movel([0.522037, -1.411516, -2.544389, -0.756484, 1.570796, 2.092833],accel_mss,speed_ms,0,blend_radius_m)
    |   movel([0.519753, -1.412609, -2.543566, -0.756214, 1.570796, 2.090549],accel_mss,speed_ms,0,blend_radius_m)
    |   movel([0.517497, -1.413267, -2.543069, -0.756052, 1.570796, 2.088293],accel_mss,speed_ms,0,blend_radius_m)
    |   movel([0.515310, -1.413576, -2.542836, -0.755977, 1.570796, 2.086106],accel_mss,speed_ms,0,blend_radius_m)
    |   movel([0.513244, -1.413623, -2.542801, -0.755965, 1.570796, 2.084041],accel_mss,speed_ms,0,blend_radius_m)
    |   movel([0.508414, -1.413136, -2.543169, -0.756085, 1.570796, 2.079211],accel_mss,speed_ms,0,blend_radius_m)
    |   movel([0.503828, -1.412721, -2.543481, -0.756187, 1.570796, 2.074625],accel_mss,speed_ms,0,blend_radius_m)
    |   movel([0.501942, -1.412771, -2.543444, -0.756174, 1.570796, 2.072738],accel_mss,speed_ms,0,blend_radius_m)
    |   movel([0.499976, -1.413061, -2.543225, -0.756103, 1.570796, 2.070772],accel_mss,speed_ms,0,blend_radius_m)
    |   movel([0.497984, -1.413655, -2.542777, -0.755957, 1.570796, 2.068780],accel_mss,speed_ms,0,blend_radius_m)
    |   movel([0.496027, -1.414618, -2.542049, -0.755723, 1.570796, 2.066824],accel_mss,speed_ms,0,blend_radius_m)
    |   movel([0.496323, -1.415340, -2.541501, -0.755547, 1.570796, 2.067119],accel_mss,speed_ms,0,blend_radius_m)
    |   movel([0.497281, -1.417258, -2.540045, -0.755086, 1.570796, 2.068077],accel_mss,speed_ms,0,blend_radius_m)
    |   movel([0.498406, -1.418772, -2.538892, -0.754725, 1.570796, 2.069203],accel_mss,speed_ms,0,blend_radius_m)
    |   movel([0.499699, -1.419880, -2.538046, -0.754464, 1.570796, 2.070495],accel_mss,speed_ms,0,blend_radius_m)
    |   movel([0.501162, -1.420584, -2.537507, -0.754298, 1.570796, 2.071959],accel_mss,speed_ms,0,blend_radius_m)
    |   movel([0.502754, -1.420928, -2.537243, -0.754218, 1.570796, 2.073551],accel_mss,speed_ms,0,blend_radius_m)
    |   movel([0.504429, -1.420952, -2.537225, -0.754212, 1.570796, 2.075225],accel_mss,speed_ms,0,blend_radius_m)
    |   movel([0.506194, -1.420656, -2.537451, -0.754281, 1.570796, 2.076990],accel_mss,speed_ms,0,blend_radius_m)
    |   movel([0.508047, -1.420040, -2.537923, -0.754426, 1.570796, 2.078844],accel_mss,speed_ms,0,blend_radius_m)
    |   movel([0.499242, -1.425154, -2.533992, -0.753243, 1.570796, 2.070038],accel_mss,speed_ms,0,blend_radius_m)
    |   movel([0.491288, -1.405893, -2.548595, -0.757901, 1.570796, 2.062085],accel_mss,speed_ms,0,blend_radius_m)
    |   movel([0.492183, -1.405355, -2.548996, -0.758039, 1.570796, 2.062980],accel_mss,speed_ms,0,blend_radius_m)
    |   speed_ms = 0.003
    |   movel([0.492183, -1.399008, -2.546063, -0.767317, 1.570796, 2.062980],accel_mss,speed_ms,0,blend_radius_m)
    |   speed_ms = 0.05
    |   movel([0.492183, -1.374535, -2.534046, -0.803807, 1.570796, 2.062980],accel_mss,speed_ms,0,blend_radius_m)
    |   #M_RunCode9
    |   movel([0.505685, -1.394015, -2.519960, -0.798414, 1.570796, 2.076481],accel_mss,speed_ms,0,blend_radius_m)
    |   #M_RunCode3
    |   movel([0.505685, -1.418115, -2.531735, -0.762539, 1.570796, 2.076481],accel_mss,speed_ms,0,blend_radius_m)
    |   speed_ms = 0.003
    |   movel([0.505685, -1.424358, -2.534606, -0.753424, 1.570796, 2.076481],accel_mss,speed_ms,0,blend_radius_m)
    |   speed_ms = 0.02
    |   movel([0.507343, -1.423678, -2.535131, -0.753580, 1.570796, 2.078139],accel_mss,speed_ms,0,blend_radius_m)
    |   movel([0.508789, -1.423672, -2.535136, -0.753582, 1.570796, 2.079585],accel_mss,speed_ms,0,blend_radius_m)
    |   movel([0.509918, -1.424231, -2.534705, -0.753454, 1.570796, 2.080714],accel_mss,speed_ms,0,blend_radius_m)
    |   movel([0.510614, -1.425248, -2.533920, -0.753222, 1.570796, 2.081410],accel_mss,speed_ms,0,blend_radius_m)
    |   movel([0.510814, -1.426544, -2.532917, -0.752928, 1.570796, 2.081610],accel_mss,speed_ms,0,blend_radius_m)
    |   movel([0.510452, -1.427953, -2.531824, -0.752612, 1.570796, 2.081249],accel_mss,speed_ms,0,blend_radius_m)
    |   movel([0.509538, -1.429300, -2.530776, -0.752313, 1.570796, 2.080334],accel_mss,speed_ms,0,blend_radius_m)
    |   movel([0.508067, -1.430415, -2.529908, -0.752067, 1.570796, 2.078864],accel_mss,speed_ms,0,blend_radius_m)
    |   movel([0.506703, -1.431026, -2.529430, -0.751933, 1.570796, 2.077499],accel_mss,speed_ms,0,blend_radius_m)
    |   movel([0.505574, -1.431213, -2.529284, -0.751892, 1.570796, 2.076370],accel_mss,speed_ms,0,blend_radius_m)
    |   movel([0.504412, -1.431493, -2.529065, -0.751831, 1.570796, 2.075208],accel_mss,speed_ms,0,blend_radius_m)
    |   movel([0.503766, -1.432035, -2.528641, -0.751713, 1.570796, 2.074562],accel_mss,speed_ms,0,blend_radius_m)
    |   movel([0.503353, -1.432783, -2.528055, -0.751551, 1.570796, 2.074150],accel_mss,speed_ms,0,blend_radius_m)
    |   movel([0.503206, -1.433607, -2.527409, -0.751373, 1.570796, 2.074002],accel_mss,speed_ms,0,blend_radius_m)
    |   movel([0.503356, -1.434381, -2.526800, -0.751208, 1.570796, 2.074152],accel_mss,speed_ms,0,blend_radius_m)
    |   movel([0.503856, -1.435229, -2.526133, -0.751027, 1.570796, 2.074653],accel_mss,speed_ms,0,blend_radius_m)
    |   movel([0.504583, -1.435849, -2.525645, -0.750896, 1.570796, 2.075379],accel_mss,speed_ms,0,blend_radius_m)
    |   movel([0.505535, -1.436238, -2.525338, -0.750814, 1.570796, 2.076331],accel_mss,speed_ms,0,blend_radius_m)
    |   movel([0.506718, -1.436396, -2.525213, -0.750780, 1.570796, 2.077514],accel_mss,speed_ms,0,blend_radius_m)
    |   movel([0.508056, -1.436320, -2.525273, -0.750796, 1.570796, 2.078852],accel_mss,speed_ms,0,blend_radius_m)
    |   movel([0.509486, -1.435996, -2.525528, -0.750865, 1.570796, 2.080282],accel_mss,speed_ms,0,blend_radius_m)
    |   movel([0.511004, -1.435426, -2.525978, -0.750985, 1.570796, 2.081801],accel_mss,speed_ms,0,blend_radius_m)
    |   movel([0.512618, -1.434610, -2.526620, -0.751159, 1.570796, 2.083414],accel_mss,speed_ms,0,blend_radius_m)
    |   movel([0.515148, -1.432826, -2.528022, -0.751542, 1.570796, 2.085945],accel_mss,speed_ms,0,blend_radius_m)
    |   movel([0.517198, -1.430614, -2.529752, -0.752023, 1.570796, 2.087995],accel_mss,speed_ms,0,blend_radius_m)
    |   movel([0.518018, -1.429355, -2.530734, -0.752300, 1.570796, 2.088814],accel_mss,speed_ms,0,blend_radius_m)
    |   movel([0.518663, -1.428007, -2.531782, -0.752600, 1.570796, 2.089459],accel_mss,speed_ms,0,blend_radius_m)
    |   movel([0.519439, -1.425040, -2.534080, -0.753269, 1.570796, 2.090235],accel_mss,speed_ms,0,blend_radius_m)
    |   movel([0.519436, -1.421793, -2.536580, -0.754016, 1.570796, 2.090232],accel_mss,speed_ms,0,blend_radius_m)
    |   movel([0.518555, -1.418352, -2.539212, -0.754825, 1.570796, 2.089351],accel_mss,speed_ms,0,blend_radius_m)
    |   movel([0.532257, -1.410606, -2.545073, -0.756710, 1.570796, 2.103054],accel_mss,speed_ms,0,blend_radius_m)
    |   movel([0.537415, -1.425473, -2.533745, -0.753170, 1.570796, 2.108212],accel_mss,speed_ms,0,blend_radius_m)
    |   movel([0.528594, -1.430343, -2.529963, -0.752083, 1.570796, 2.099390],accel_mss,speed_ms,0,blend_radius_m)
    |   movel([0.530498, -1.428621, -2.531305, -0.752463, 1.570796, 2.101294],accel_mss,speed_ms,0,blend_radius_m)
    |   movel([0.532054, -1.426533, -2.532925, -0.752931, 1.570796, 2.102850],accel_mss,speed_ms,0,blend_radius_m)
    |   movel([0.533176, -1.424184, -2.534740, -0.753464, 1.570796, 2.103972],accel_mss,speed_ms,0,blend_radius_m)
    |   movel([0.533790, -1.421674, -2.536671, -0.754044, 1.570796, 2.104586],accel_mss,speed_ms,0,blend_radius_m)
    |   movel([0.533838, -1.419100, -2.538642, -0.754648, 1.570796, 2.104634],accel_mss,speed_ms,0,blend_radius_m)
    |   movel([0.533270, -1.416566, -2.540572, -0.755252, 1.570796, 2.104066],accel_mss,speed_ms,0,blend_radius_m)
    |   movel([0.523200, -1.422207, -2.536262, -0.753920, 1.570796, 2.093996],accel_mss,speed_ms,0,blend_radius_m)
    |   movel([0.523982, -1.425264, -2.533907, -0.753218, 1.570796, 2.094778],accel_mss,speed_ms,0,blend_radius_m)
    |   movel([0.524165, -1.428496, -2.531402, -0.752491, 1.570796, 2.094961],accel_mss,speed_ms,0,blend_radius_m)
    |   movel([0.523653, -1.431730, -2.528880, -0.751779, 1.570796, 2.094449],accel_mss,speed_ms,0,blend_radius_m)
    |   movel([0.523103, -1.433286, -2.527660, -0.751442, 1.570796, 2.093899],accel_mss,speed_ms,0,blend_radius_m)
    |   movel([0.522353, -1.434804, -2.526468, -0.751117, 1.570796, 2.093149],accel_mss,speed_ms,0,blend_radius_m)
    |   movel([0.521392, -1.436236, -2.525339, -0.750814, 1.570796, 2.092189],accel_mss,speed_ms,0,blend_radius_m)
    |   movel([0.520203, -1.437537, -2.524311, -0.750541, 1.570796, 2.090999],accel_mss,speed_ms,0,blend_radius_m)
    |   movel([0.518786, -1.438713, -2.523380, -0.750296, 1.570796, 2.089582],accel_mss,speed_ms,0,blend_radius_m)
    |   movel([0.517140, -1.439760, -2.522548, -0.750080, 1.570796, 2.087936],accel_mss,speed_ms,0,blend_radius_m)
    |   movel([0.515419, -1.440606, -2.521876, -0.749907, 1.570796, 2.086215],accel_mss,speed_ms,0,blend_radius_m)
    |   movel([0.513770, -1.441178, -2.521420, -0.749790, 1.570796, 2.084567],accel_mss,speed_ms,0,blend_radius_m)
    |   movel([0.512194, -1.441476, -2.521183, -0.749730, 1.570796, 2.082991],accel_mss,speed_ms,0,blend_radius_m)
    |   movel([0.510687, -1.441499, -2.521165, -0.749725, 1.570796, 2.081483],accel_mss,speed_ms,0,blend_radius_m)
    |   movel([0.507968, -1.440895, -2.521646, -0.749848, 1.570796, 2.078764],accel_mss,speed_ms,0,blend_radius_m)
    |   movel([0.505701, -1.439532, -2.522730, -0.750127, 1.570796, 2.076497],accel_mss,speed_ms,0,blend_radius_m)
    |   movel([0.503914, -1.437597, -2.524264, -0.750528, 1.570796, 2.074711],accel_mss,speed_ms,0,blend_radius_m)
    |   movel([0.502646, -1.435274, -2.526097, -0.751017, 1.570796, 2.073442],accel_mss,speed_ms,0,blend_radius_m)
    |   movel([0.502142, -1.433468, -2.527518, -0.751403, 1.570796, 2.072938],accel_mss,speed_ms,0,blend_radius_m)
    |   movel([0.501979, -1.431437, -2.529109, -0.751843, 1.570796, 2.072776],accel_mss,speed_ms,0,blend_radius_m)
    |   movel([0.502213, -1.429345, -2.530741, -0.752303, 1.570796, 2.073009],accel_mss,speed_ms,0,blend_radius_m)
    |   movel([0.502903, -1.427364, -2.532281, -0.752744, 1.570796, 2.073699],accel_mss,speed_ms,0,blend_radius_m)
    |   movel([0.504056, -1.425650, -2.533608, -0.753130, 1.570796, 2.074852],accel_mss,speed_ms,0,blend_radius_m)
    |   movel([0.505685, -1.424358, -2.534606, -0.753424, 1.570796, 2.076481],accel_mss,speed_ms,0,blend_radius_m)
    |   speed_ms = 0.003
    |   movel([0.505685, -1.418115, -2.531735, -0.762539, 1.570796, 2.076481],accel_mss,speed_ms,0,blend_radius_m)
    |   speed_ms = 0.05
    |   movel([0.505685, -1.394015, -2.519960, -0.798414, 1.570796, 2.076481],accel_mss,speed_ms,0,blend_radius_m)
    |   #M_RunCode9
    |   movel([0.511765, -1.313908, -2.574588, -0.823893, 1.570796, 2.082561],accel_mss,speed_ms,0,blend_radius_m)
    |   #M_RunCode3
    |   movel([0.511765, -1.339451, -2.587378, -0.785560, 1.570796, 2.082561],accel_mss,speed_ms,0,blend_radius_m)
    |   speed_ms = 0.003
    |   movel([0.511765, -1.346101, -2.590505, -0.775783, 1.570796, 2.082561],accel_mss,speed_ms,0,blend_radius_m)
    |   speed_ms = 0.02
    |   movel([0.509003, -1.346634, -2.590154, -0.775602, 1.570796, 2.079799],accel_mss,speed_ms,0,blend_radius_m)
    |   movel([0.506323, -1.346604, -2.590173, -0.775612, 1.570796, 2.077120],accel_mss,speed_ms,0,blend_radius_m)
    |   movel([0.503779, -1.346109, -2.590499, -0.775781, 1.570796, 2.074576],accel_mss,speed_ms,0,blend_radius_m)
    |   movel([0.501429, -1.345241, -2.591071, -0.776077, 1.570796, 2.072225],accel_mss,speed_ms,0,blend_radius_m)
    |   movel([0.499334, -1.344090, -2.591827, -0.776472, 1.570796, 2.070130],accel_mss,speed_ms,0,blend_radius_m)
    |   movel([0.500903, -1.340898, -2.593914, -0.777577, 1.570796, 2.071699],accel_mss,speed_ms,0,blend_radius_m)
    |   movel([0.503381, -1.337486, -2.596130, -0.778773, 1.570796, 2.074177],accel_mss,speed_ms,0,blend_radius_m)
    |   movel([0.506519, -1.334154, -2.598278, -0.779957, 1.570796, 2.077315],accel_mss,speed_ms,0,blend_radius_m)
    |   movel([0.510041, -1.331225, -2.600155, -0.781010, 1.570796, 2.080838],accel_mss,speed_ms,0,blend_radius_m)
    |   movel([0.513677, -1.329019, -2.601560, -0.781810, 1.570796, 2.084474],accel_mss,speed_ms,0,blend_radius_m)
    |   movel([0.515448, -1.328288, -2.602024, -0.782077, 1.570796, 2.086244],accel_mss,speed_ms,0,blend_radius_m)
    |   movel([0.517140, -1.327859, -2.602297, -0.782234, 1.570796, 2.087936],accel_mss,speed_ms,0,blend_radius_m)
    |   movel([0.518717, -1.327772, -2.602352, -0.782265, 1.570796, 2.089514],accel_mss,speed_ms,0,blend_radius_m)
    |   movel([0.520146, -1.328066, -2.602165, -0.782158, 1.570796, 2.090942],accel_mss,speed_ms,0,blend_radius_m)
    |   movel([0.521388, -1.328777, -2.601714, -0.781898, 1.570796, 2.092184],accel_mss,speed_ms,0,blend_radius_m)
    |   movel([0.522405, -1.329948, -2.600969, -0.781472, 1.570796, 2.093201],accel_mss,speed_ms,0,blend_radius_m)
    |   movel([0.523173, -1.332184, -2.599542, -0.780663, 1.570796, 2.093970],accel_mss,speed_ms,0,blend_radius_m)
    |   movel([0.522946, -1.334699, -2.597928, -0.779762, 1.570796, 2.093742],accel_mss,speed_ms,0,blend_radius_m)
    |   movel([0.521842, -1.337390, -2.596192, -0.778807, 1.570796, 2.092638],accel_mss,speed_ms,0,blend_radius_m)
    |   movel([0.519982, -1.340150, -2.594401, -0.777838, 1.570796, 2.090778],accel_mss,speed_ms,0,blend_radius_m)
    |   movel([0.517307, -1.342963, -2.592565, -0.776861, 1.570796, 2.088104],accel_mss,speed_ms,0,blend_radius_m)
    |   movel([0.514551, -1.344910, -2.591288, -0.776190, 1.570796, 2.085348],accel_mss,speed_ms,0,blend_radius_m)
    |   movel([0.511765, -1.346101, -2.590505, -0.775783, 1.570796, 2.082561],accel_mss,speed_ms,0,blend_radius_m)
    |   speed_ms = 0.003
    |   movel([0.511765, -1.339451, -2.587378, -0.785560, 1.570796, 2.082561],accel_mss,speed_ms,0,blend_radius_m)
    |   speed_ms = 0.05
    |   movel([0.511765, -1.313908, -2.574588, -0.823893, 1.570796, 2.082561],accel_mss,speed_ms,0,blend_radius_m)
    |   #M_RunCode9
    |   movel([0.593175, -1.228303, -2.623878, -0.860208, 1.570796, 2.163971],accel_mss,speed_ms,0,blend_radius_m)
    |   #M_RunCode3
    |   movel([0.593175, -1.255054, -2.637790, -0.819545, 1.570796, 2.163971],accel_mss,speed_ms,0,blend_radius_m)
    |   speed_ms = 0.003
    |   movel([0.593175, -1.262061, -2.641200, -0.809128, 1.570796, 2.163971],accel_mss,speed_ms,0,blend_radius_m)
    |   speed_ms = 0.02
    |   movel([0.592118, -1.260949, -2.641811, -0.809629, 1.570796, 2.162914],accel_mss,speed_ms,0,blend_radius_m)
    |   movel([0.591505, -1.259430, -2.642643, -0.810317, 1.570796, 2.162302],accel_mss,speed_ms,0,blend_radius_m)
    |   movel([0.591148, -1.257700, -2.643586, -0.811103, 1.570796, 2.161944],accel_mss,speed_ms,0,blend_radius_m)
    |   movel([0.591952, -1.257478, -2.643707, -0.811204, 1.570796, 2.162749],accel_mss,speed_ms,0,blend_radius_m)
    |   movel([0.592411, -1.257816, -2.643523, -0.811050, 1.570796, 2.163207],accel_mss,speed_ms,0,blend_radius_m)
    |   movel([0.592987, -1.258156, -2.643338, -0.810895, 1.570796, 2.163783],accel_mss,speed_ms,0,blend_radius_m)
    |   movel([0.594138, -1.257945, -2.643453, -0.810991, 1.570796, 2.164934],accel_mss,speed_ms,0,blend_radius_m)
    |   movel([0.595427, -1.257217, -2.643850, -0.811323, 1.570796, 2.166224],accel_mss,speed_ms,0,blend_radius_m)
    |   movel([0.596669, -1.256262, -2.644368, -0.811759, 1.570796, 2.167466],accel_mss,speed_ms,0,blend_radius_m)
    |   movel([0.598371, -1.254882, -2.645116, -0.812391, 1.570796, 2.169167],accel_mss,speed_ms,0,blend_radius_m)
    |   movel([0.598070, -1.252620, -2.646337, -0.813432, 1.570796, 2.168867],accel_mss,speed_ms,0,blend_radius_m)
    |   movel([0.597149, -1.251145, -2.647130, -0.814114, 1.570796, 2.167945],accel_mss,speed_ms,0,blend_radius_m)
    |   movel([0.596399, -1.250811, -2.647309, -0.814269, 1.570796, 2.167195],accel_mss,speed_ms,0,blend_radius_m)
    |   movel([0.595425, -1.250808, -2.647311, -0.814270, 1.570796, 2.166221],accel_mss,speed_ms,0,blend_radius_m)
    |   movel([0.594204, -1.251181, -2.647110, -0.814097, 1.570796, 2.165000],accel_mss,speed_ms,0,blend_radius_m)
    |   movel([0.592717, -1.251976, -2.646684, -0.813730, 1.570796, 2.163513],accel_mss,speed_ms,0,blend_radius_m)
    |   movel([0.593308, -1.250419, -2.647519, -0.814451, 1.570796, 2.164105],accel_mss,speed_ms,0,blend_radius_m)
    |   movel([0.593995, -1.249081, -2.648235, -0.815073, 1.570796, 2.164792],accel_mss,speed_ms,0,blend_radius_m)
    |   movel([0.594412, -1.248607, -2.648488, -0.815294, 1.570796, 2.165208],accel_mss,speed_ms,0,blend_radius_m)
    |   movel([0.594899, -1.248328, -2.648637, -0.815424, 1.570796, 2.165695],accel_mss,speed_ms,0,blend_radius_m)
    |   movel([0.596139, -1.248534, -2.648527, -0.815328, 1.570796, 2.166935],accel_mss,speed_ms,0,blend_radius_m)
    |   movel([0.597985, -1.249993, -2.647747, -0.814649, 1.570796, 2.168781],accel_mss,speed_ms,0,blend_radius_m)
    |   movel([0.599239, -1.252067, -2.646635, -0.813688, 1.570796, 2.170035],accel_mss,speed_ms,0,blend_radius_m)
    |   movel([0.599500, -1.253288, -2.645977, -0.813124, 1.570796, 2.170297],accel_mss,speed_ms,0,blend_radius_m)
    |   movel([0.599438, -1.254612, -2.645262, -0.812515, 1.570796, 2.170234],accel_mss,speed_ms,0,blend_radius_m)
    |   movel([0.598999, -1.256018, -2.644501, -0.811870, 1.570796, 2.169795],accel_mss,speed_ms,0,blend_radius_m)
    |   movel([0.598125, -1.257489, -2.643701, -0.811199, 1.570796, 2.168921],accel_mss,speed_ms,0,blend_radius_m)
    |   movel([0.596913, -1.256631, -2.644168, -0.811590, 1.570796, 2.167709],accel_mss,speed_ms,0,blend_radius_m)
    |   movel([0.594869, -1.262559, -2.640926, -0.808904, 1.570796, 2.165665],accel_mss,speed_ms,0,blend_radius_m)
    |   movel([0.593175, -1.262061, -2.641200, -0.809128, 1.570796, 2.163971],accel_mss,speed_ms,0,blend_radius_m)
    |   speed_ms = 0.003
    |   movel([0.593175, -1.255054, -2.637790, -0.819545, 1.570796, 2.163971],accel_mss,speed_ms,0,blend_radius_m)
    |   speed_ms = 0.05
    |   movel([0.593175, -1.228303, -2.623878, -0.860208, 1.570796, 2.163971],accel_mss,speed_ms,0,blend_radius_m)
    |   #M_RunCode9
    |   movel([0.574585, -1.187672, -2.644287, -0.880430, 1.570796, 2.145381],accel_mss,speed_ms,0,blend_radius_m)
    |   #M_RunCode3
    |   movel([0.574585, -1.214836, -2.658735, -0.838818, 1.570796, 2.145381],accel_mss,speed_ms,0,blend_radius_m)
    |   speed_ms = 0.003
    |   movel([0.574585, -1.221975, -2.662282, -0.828132, 1.570796, 2.145381],accel_mss,speed_ms,0,blend_radius_m)
    |   speed_ms = 0.02
    |   movel([0.571968, -1.223903, -2.661311, -0.827175, 1.570796, 2.142764],accel_mss,speed_ms,0,blend_radius_m)
    |   movel([0.569236, -1.225606, -2.660449, -0.826333, 1.570796, 2.140032],accel_mss,speed_ms,0,blend_radius_m)
    |   movel([0.566418, -1.227048, -2.659718, -0.825623, 1.570796, 2.137214],accel_mss,speed_ms,0,blend_radius_m)
    |   movel([0.563541, -1.228201, -2.659131, -0.825057, 1.570796, 2.134337],accel_mss,speed_ms,0,blend_radius_m)
    |   movel([0.560640, -1.229035, -2.658705, -0.824649, 1.570796, 2.131436],accel_mss,speed_ms,0,blend_radius_m)
    |   movel([0.559180, -1.229158, -2.658643, -0.824589, 1.570796, 2.129976],accel_mss,speed_ms,0,blend_radius_m)
    |   movel([0.557735, -1.229044, -2.658701, -0.824644, 1.570796, 2.128531],accel_mss,speed_ms,0,blend_radius_m)
    |   movel([0.556429, -1.228954, -2.658747, -0.824688, 1.570796, 2.127225],accel_mss,speed_ms,0,blend_radius_m)
    |   movel([0.555404, -1.229136, -2.658654, -0.824599, 1.570796, 2.126200],accel_mss,speed_ms,0,blend_radius_m)
    |   movel([0.553651, -1.230355, -2.658030, -0.824004, 1.570796, 2.124447],accel_mss,speed_ms,0,blend_radius_m)
    |   movel([0.551341, -1.232324, -2.657020, -0.823045, 1.570796, 2.122138],accel_mss,speed_ms,0,blend_radius_m)
    |   movel([0.548946, -1.234404, -2.655947, -0.822038, 1.570796, 2.119742],accel_mss,speed_ms,0,blend_radius_m)
    |   movel([0.546922, -1.235960, -2.655141, -0.821287, 1.570796, 2.117718],accel_mss,speed_ms,0,blend_radius_m)
    |   movel([0.542914, -1.238247, -2.653952, -0.820190, 1.570796, 2.113711],accel_mss,speed_ms,0,blend_radius_m)
    |   movel([0.539333, -1.239717, -2.653184, -0.819487, 1.570796, 2.110130],accel_mss,speed_ms,0,blend_radius_m)
    |   movel([0.536136, -1.240454, -2.652799, -0.819136, 1.570796, 2.106932],accel_mss,speed_ms,0,blend_radius_m)
    |   movel([0.533287, -1.240532, -2.652758, -0.819099, 1.570796, 2.104083],accel_mss,speed_ms,0,blend_radius_m)
    |   movel([0.530754, -1.240029, -2.653021, -0.819339, 1.570796, 2.101551],accel_mss,speed_ms,0,blend_radius_m)
    |   movel([0.528507, -1.239015, -2.653552, -0.819823, 1.570796, 2.099304],accel_mss,speed_ms,0,blend_radius_m)
    |   movel([0.526515, -1.237561, -2.654309, -0.820518, 1.570796, 2.097311],accel_mss,speed_ms,0,blend_radius_m)
    |   movel([0.524746, -1.235741, -2.655255, -0.821393, 1.570796, 2.095543],accel_mss,speed_ms,0,blend_radius_m)
    |   movel([0.521770, -1.231289, -2.657552, -0.823549, 1.570796, 2.092567],accel_mss,speed_ms,0,blend_radius_m)
    |   movel([0.519363, -1.226237, -2.660130, -0.826023, 1.570796, 2.090159],accel_mss,speed_ms,0,blend_radius_m)
    |   movel([0.515384, -1.216730, -2.664902, -0.830757, 1.570796, 2.086180],accel_mss,speed_ms,0,blend_radius_m)
    |   movel([0.513122, -1.212916, -2.666788, -0.832686, 1.570796, 2.083919],accel_mss,speed_ms,0,blend_radius_m)
    |   movel([0.509996, -1.208909, -2.668751, -0.834729, 1.570796, 2.080792],accel_mss,speed_ms,0,blend_radius_m)
    |   movel([0.506128, -1.204957, -2.670670, -0.836762, 1.570796, 2.076924],accel_mss,speed_ms,0,blend_radius_m)
    |   movel([0.501653, -1.201305, -2.672428, -0.838656, 1.570796, 2.072450],accel_mss,speed_ms,0,blend_radius_m)
    |   movel([0.496713, -1.198205, -2.673909, -0.840275, 1.570796, 2.067510],accel_mss,speed_ms,0,blend_radius_m)
    |   movel([0.491464, -1.195895, -2.675005, -0.841489, 1.570796, 2.062260],accel_mss,speed_ms,0,blend_radius_m)
    |   movel([0.486068, -1.194615, -2.675610, -0.842164, 1.570796, 2.056864],accel_mss,speed_ms,0,blend_radius_m)
    |   movel([0.483368, -1.194435, -2.675696, -0.842259, 1.570796, 2.054164],accel_mss,speed_ms,0,blend_radius_m)
    |   movel([0.480698, -1.194593, -2.675621, -0.842175, 1.570796, 2.051494],accel_mss,speed_ms,0,blend_radius_m)
    |   movel([0.477824, -1.195119, -2.675372, -0.841897, 1.570796, 2.048620],accel_mss,speed_ms,0,blend_radius_m)
    |   movel([0.474379, -1.196066, -2.674924, -0.841399, 1.570796, 2.045175],accel_mss,speed_ms,0,blend_radius_m)
    |   movel([0.470557, -1.197461, -2.674262, -0.840665, 1.570796, 2.041354],accel_mss,speed_ms,0,blend_radius_m)
    |   movel([0.466556, -1.199323, -2.673376, -0.839690, 1.570796, 2.037353],accel_mss,speed_ms,0,blend_radius_m)
    |   movel([0.462584, -1.201663, -2.672256, -0.838470, 1.570796, 2.033380],accel_mss,speed_ms,0,blend_radius_m)
    |   movel([0.458831, -1.204496, -2.670893, -0.837000, 1.570796, 2.029628],accel_mss,speed_ms,0,blend_radius_m)
    |   movel([0.455502, -1.207831, -2.669276, -0.835282, 1.570796, 2.026298],accel_mss,speed_ms,0,blend_radius_m)
    |   movel([0.454056, -1.209685, -2.668372, -0.834332, 1.570796, 2.024852],accel_mss,speed_ms,0,blend_radius_m)
    |   movel([0.452789, -1.211669, -2.667401, -0.833320, 1.570796, 2.023586],accel_mss,speed_ms,0,blend_radius_m)
    |   movel([0.451398, -1.214773, -2.665871, -0.831745, 1.570796, 2.022194],accel_mss,speed_ms,0,blend_radius_m)
    |   movel([0.450982, -1.217407, -2.664565, -0.830417, 1.570796, 2.021778],accel_mss,speed_ms,0,blend_radius_m)
    |   movel([0.451430, -1.219618, -2.663463, -0.829308, 1.570796, 2.022226],accel_mss,speed_ms,0,blend_radius_m)
    |   movel([0.452634, -1.221449, -2.662546, -0.828394, 1.570796, 2.023430],accel_mss,speed_ms,0,blend_radius_m)
    |   movel([0.454488, -1.222942, -2.661795, -0.827652, 1.570796, 2.025284],accel_mss,speed_ms,0,blend_radius_m)
    |   movel([0.456887, -1.224143, -2.661190, -0.827057, 1.570796, 2.027683],accel_mss,speed_ms,0,blend_radius_m)
    |   movel([0.459731, -1.225090, -2.660711, -0.826588, 1.570796, 2.030527],accel_mss,speed_ms,0,blend_radius_m)
    |   movel([0.462914, -1.225829, -2.660337, -0.826224, 1.570796, 2.033710],accel_mss,speed_ms,0,blend_radius_m)
    |   movel([0.469896, -1.226823, -2.659832, -0.825734, 1.570796, 2.040692],accel_mss,speed_ms,0,blend_radius_m)
    |   movel([0.477036, -1.227418, -2.659530, -0.825442, 1.570796, 2.047832],accel_mss,speed_ms,0,blend_radius_m)
    |   movel([0.483538, -1.227875, -2.659297, -0.825217, 1.570796, 2.054334],accel_mss,speed_ms,0,blend_radius_m)
    |   movel([0.488608, -1.228447, -2.659005, -0.824936, 1.570796, 2.059404],accel_mss,speed_ms,0,blend_radius_m)
    |   movel([0.500502, -1.230472, -2.657970, -0.823947, 1.570796, 2.071299],accel_mss,speed_ms,0,blend_radius_m)
    |   movel([0.506711, -1.231796, -2.657291, -0.823302, 1.570796, 2.077507],accel_mss,speed_ms,0,blend_radius_m)
    |   movel([0.511317, -1.233209, -2.656564, -0.822616, 1.570796, 2.082113],accel_mss,speed_ms,0,blend_radius_m)
    |   movel([0.512898, -1.234063, -2.656123, -0.822203, 1.570796, 2.083694],accel_mss,speed_ms,0,blend_radius_m)
    |   movel([0.514219, -1.235153, -2.655560, -0.821676, 1.570796, 2.085015],accel_mss,speed_ms,0,blend_radius_m)
    |   movel([0.516112, -1.237960, -2.654102, -0.820327, 1.570796, 2.086908],accel_mss,speed_ms,0,blend_radius_m)
    |   movel([0.517083, -1.241449, -2.652277, -0.818663, 1.570796, 2.087879],accel_mss,speed_ms,0,blend_radius_m)
    |   movel([0.517232, -1.245433, -2.650175, -0.816780, 1.570796, 2.088029],accel_mss,speed_ms,0,blend_radius_m)
    |   movel([0.516645, -1.249736, -2.647885, -0.814768, 1.570796, 2.087441],accel_mss,speed_ms,0,blend_radius_m)
    |   movel([0.515414, -1.254188, -2.645491, -0.812710, 1.570796, 2.086210],accel_mss,speed_ms,0,blend_radius_m)
    |   movel([0.513627, -1.258624, -2.643083, -0.810682, 1.570796, 2.084424],accel_mss,speed_ms,0,blend_radius_m)
    |   movel([0.511373, -1.262878, -2.640751, -0.808760, 1.570796, 2.082169],accel_mss,speed_ms,0,blend_radius_m)
    |   movel([0.507975, -1.267863, -2.637990, -0.806536, 1.570796, 2.078771],accel_mss,speed_ms,0,blend_radius_m)
    |   movel([0.506300, -1.269831, -2.636892, -0.805667, 1.570796, 2.077097],accel_mss,speed_ms,0,blend_radius_m)
    |   movel([0.504622, -1.271495, -2.635959, -0.804935, 1.570796, 2.075419],accel_mss,speed_ms,0,blend_radius_m)
    |   movel([0.502938, -1.272892, -2.635173, -0.804323, 1.570796, 2.073734],accel_mss,speed_ms,0,blend_radius_m)
    |   movel([0.501232, -1.274054, -2.634518, -0.803816, 1.570796, 2.072029],accel_mss,speed_ms,0,blend_radius_m)
    |   movel([0.497721, -1.275822, -2.633518, -0.803049, 1.570796, 2.068517],accel_mss,speed_ms,0,blend_radius_m)
    |   movel([0.494012, -1.277065, -2.632813, -0.802511, 1.570796, 2.064808],accel_mss,speed_ms,0,blend_radius_m)
    |   movel([0.490033, -1.278049, -2.632253, -0.802087, 1.570796, 2.060830],accel_mss,speed_ms,0,blend_radius_m)
    |   movel([0.480997, -1.280279, -2.630980, -0.801130, 1.570796, 2.051793],accel_mss,speed_ms,0,blend_radius_m)
    |   movel([0.480527, -1.280438, -2.630889, -0.801062, 1.570796, 2.051324],accel_mss,speed_ms,0,blend_radius_m)
    |   movel([0.480674, -1.280531, -2.630836, -0.801023, 1.570796, 2.051471],accel_mss,speed_ms,0,blend_radius_m)
    |   movel([0.482495, -1.280556, -2.630822, -0.801012, 1.570796, 2.053291],accel_mss,speed_ms,0,blend_radius_m)
    |   movel([0.489992, -1.280226, -2.631010, -0.801153, 1.570796, 2.060788],accel_mss,speed_ms,0,blend_radius_m)
    |   movel([0.502407, -1.279760, -2.631277, -0.801352, 1.570796, 2.073204],accel_mss,speed_ms,0,blend_radius_m)
    |   movel([0.495040, -1.283177, -2.629316, -0.799896, 1.570796, 2.065836],accel_mss,speed_ms,0,blend_radius_m)
    |   movel([0.486849, -1.286617, -2.627328, -0.798445, 1.570796, 2.057645],accel_mss,speed_ms,0,blend_radius_m)
    |   movel([0.478134, -1.290012, -2.625350, -0.797027, 1.570796, 2.048930],accel_mss,speed_ms,0,blend_radius_m)
    |   movel([0.469185, -1.293284, -2.623430, -0.795675, 1.570796, 2.039981],accel_mss,speed_ms,0,blend_radius_m)
    |   movel([0.451739, -1.299146, -2.619956, -0.793286, 1.570796, 2.022535],accel_mss,speed_ms,0,blend_radius_m)
    |   movel([0.443813, -1.301554, -2.618517, -0.792318, 1.570796, 2.014610],accel_mss,speed_ms,0,blend_radius_m)
    |   movel([0.436791, -1.303489, -2.617355, -0.791545, 1.570796, 2.007588],accel_mss,speed_ms,0,blend_radius_m)
    |   movel([0.426899, -1.309868, -2.613488, -0.789032, 1.570796, 1.997696],accel_mss,speed_ms,0,blend_radius_m)
    |   movel([0.416898, -1.316826, -2.609211, -0.786352, 1.570796, 1.987694],accel_mss,speed_ms,0,blend_radius_m)
    |   movel([0.396911, -1.331466, -2.600001, -0.780922, 1.570796, 1.967707],accel_mss,speed_ms,0,blend_radius_m)
    |   movel([0.387059, -1.338680, -2.595356, -0.778353, 1.570796, 1.957856],accel_mss,speed_ms,0,blend_radius_m)
    |   movel([0.377371, -1.345531, -2.590880, -0.775978, 1.570796, 1.948167],accel_mss,speed_ms,0,blend_radius_m)
    |   movel([0.367887, -1.351814, -2.586718, -0.773857, 1.570796, 1.938684],accel_mss,speed_ms,0,blend_radius_m)
    |   movel([0.358636, -1.357329, -2.583020, -0.772040, 1.570796, 1.929432],accel_mss,speed_ms,0,blend_radius_m)
    |   movel([0.355051, -1.359183, -2.581767, -0.771438, 1.570796, 1.925847],accel_mss,speed_ms,0,blend_radius_m)
    |   movel([0.351650, -1.360673, -2.580757, -0.770959, 1.570796, 1.922446],accel_mss,speed_ms,0,blend_radius_m)
    |   movel([0.348454, -1.361801, -2.579990, -0.770598, 1.570796, 1.919251],accel_mss,speed_ms,0,blend_radius_m)
    |   movel([0.345478, -1.362574, -2.579464, -0.770351, 1.570796, 1.916275],accel_mss,speed_ms,0,blend_radius_m)
    |   movel([0.342741, -1.362990, -2.579180, -0.770219, 1.570796, 1.913537],accel_mss,speed_ms,0,blend_radius_m)
    |   movel([0.340260, -1.363051, -2.579138, -0.770199, 1.570796, 1.911056],accel_mss,speed_ms,0,blend_radius_m)
    |   movel([0.338052, -1.362760, -2.579337, -0.770292, 1.570796, 1.908848],accel_mss,speed_ms,0,blend_radius_m)
    |   movel([0.336140, -1.362118, -2.579775, -0.770496, 1.570796, 1.906937],accel_mss,speed_ms,0,blend_radius_m)
    |   movel([0.334544, -1.361121, -2.580453, -0.770815, 1.570796, 1.905340],accel_mss,speed_ms,0,blend_radius_m)
    |   movel([0.333283, -1.359768, -2.581371, -0.771250, 1.570796, 1.904079],accel_mss,speed_ms,0,blend_radius_m)
    |   movel([0.332383, -1.358059, -2.582528, -0.771803, 1.570796, 1.903179],accel_mss,speed_ms,0,blend_radius_m)
    |   movel([0.331860, -1.355992, -2.583921, -0.772477, 1.570796, 1.902657],accel_mss,speed_ms,0,blend_radius_m)
    |   movel([0.331745, -1.353561, -2.585551, -0.773277, 1.570796, 1.902541],accel_mss,speed_ms,0,blend_radius_m)
    |   movel([0.332061, -1.350763, -2.587418, -0.774208, 1.570796, 1.902857],accel_mss,speed_ms,0,blend_radius_m)
    |   movel([0.332833, -1.347594, -2.589520, -0.775275, 1.570796, 1.903629],accel_mss,speed_ms,0,blend_radius_m)
    |   movel([0.334091, -1.344048, -2.591854, -0.776487, 1.570796, 1.904887],accel_mss,speed_ms,0,blend_radius_m)
    |   movel([0.336817, -1.345103, -2.591162, -0.776125, 1.570796, 1.907613],accel_mss,speed_ms,0,blend_radius_m)
    |   movel([0.338210, -1.345526, -2.590883, -0.775980, 1.570796, 1.909006],accel_mss,speed_ms,0,blend_radius_m)
    |   movel([0.339758, -1.345563, -2.590859, -0.775967, 1.570796, 1.910555],accel_mss,speed_ms,0,blend_radius_m)
    |   movel([0.341117, -1.345166, -2.591120, -0.776103, 1.570796, 1.911913],accel_mss,speed_ms,0,blend_radius_m)
    |   movel([0.342815, -1.344348, -2.591658, -0.776384, 1.570796, 1.913611],accel_mss,speed_ms,0,blend_radius_m)
    |   movel([0.347048, -1.341647, -2.593426, -0.777316, 1.570796, 1.917845],accel_mss,speed_ms,0,blend_radius_m)
    |   movel([0.352103, -1.337874, -2.595879, -0.778636, 1.570796, 1.922899],accel_mss,speed_ms,0,blend_radius_m)
    |   movel([0.357611, -1.333435, -2.598740, -0.780214, 1.570796, 1.928407],accel_mss,speed_ms,0,blend_radius_m)
    |   movel([0.368447, -1.324252, -2.604575, -0.783562, 1.570796, 1.939243],accel_mss,speed_ms,0,blend_radius_m)
    |   movel([0.376352, -1.317549, -2.608763, -0.786077, 1.570796, 1.947148],accel_mss,speed_ms,0,blend_radius_m)
    |   movel([0.383444, -1.312172, -2.612079, -0.788138, 1.570796, 1.954240],accel_mss,speed_ms,0,blend_radius_m)
    |   movel([0.390604, -1.306773, -2.615371, -0.790245, 1.570796, 1.961401],accel_mss,speed_ms,0,blend_radius_m)
    |   movel([0.376307, -1.309577, -2.613666, -0.789146, 1.570796, 1.947104],accel_mss,speed_ms,0,blend_radius_m)
    |   movel([0.368938, -1.310738, -2.612957, -0.788693, 1.570796, 1.939734],accel_mss,speed_ms,0,blend_radius_m)
    |   movel([0.361948, -1.311238, -2.612652, -0.788499, 1.570796, 1.932745],accel_mss,speed_ms,0,blend_radius_m)
    |   movel([0.358718, -1.311117, -2.612726, -0.788547, 1.570796, 1.929514],accel_mss,speed_ms,0,blend_radius_m)
    |   movel([0.355728, -1.310684, -2.612991, -0.788715, 1.570796, 1.926524],accel_mss,speed_ms,0,blend_radius_m)
    |   movel([0.353028, -1.309887, -2.613477, -0.789025, 1.570796, 1.923824],accel_mss,speed_ms,0,blend_radius_m)
    |   movel([0.350666, -1.308677, -2.614215, -0.789497, 1.570796, 1.921462],accel_mss,speed_ms,0,blend_radius_m)
    |   movel([0.348690, -1.307001, -2.615233, -0.790155, 1.570796, 1.919486],accel_mss,speed_ms,0,blend_radius_m)
    |   movel([0.347151, -1.304805, -2.616561, -0.791022, 1.570796, 1.917947],accel_mss,speed_ms,0,blend_radius_m)
    |   movel([0.346102, -1.302030, -2.618232, -0.792127, 1.570796, 1.916898],accel_mss,speed_ms,0,blend_radius_m)
    |   movel([0.345599, -1.298617, -2.620272, -0.793500, 1.570796, 1.916395],accel_mss,speed_ms,0,blend_radius_m)
    |   movel([0.345849, -1.294212, -2.622883, -0.795294, 1.570796, 1.916645],accel_mss,speed_ms,0,blend_radius_m)
    |   movel([0.347025, -1.289411, -2.625701, -0.797277, 1.570796, 1.917821],accel_mss,speed_ms,0,blend_radius_m)
    |   movel([0.349047, -1.284362, -2.628633, -0.799394, 1.570796, 1.919843],accel_mss,speed_ms,0,blend_radius_m)
    |   movel([0.351840, -1.279224, -2.631583, -0.801582, 1.570796, 1.922636],accel_mss,speed_ms,0,blend_radius_m)
    |   movel([0.355317, -1.274164, -2.634456, -0.803769, 1.570796, 1.926113],accel_mss,speed_ms,0,blend_radius_m)
    |   movel([0.359387, -1.269353, -2.637159, -0.805878, 1.570796, 1.930184],accel_mss,speed_ms,0,blend_radius_m)
    |   movel([0.363958, -1.264968, -2.639597, -0.807824, 1.570796, 1.934754],accel_mss,speed_ms,0,blend_radius_m)
    |   movel([0.368923, -1.261200, -2.641673, -0.809516, 1.570796, 1.939720],accel_mss,speed_ms,0,blend_radius_m)
    |   movel([0.371754, -1.259742, -2.642472, -0.810175, 1.570796, 1.942550],accel_mss,speed_ms,0,blend_radius_m)
    |   movel([0.374895, -1.258734, -2.643023, -0.810632, 1.570796, 1.945692],accel_mss,speed_ms,0,blend_radius_m)
    |   movel([0.377336, -1.258552, -2.643122, -0.810715, 1.570796, 1.948132],accel_mss,speed_ms,0,blend_radius_m)
    |   movel([0.377979, -1.258887, -2.642939, -0.810563, 1.570796, 1.948775],accel_mss,speed_ms,0,blend_radius_m)
    |   movel([0.378068, -1.259568, -2.642567, -0.810254, 1.570796, 1.948864],accel_mss,speed_ms,0,blend_radius_m)
    |   movel([0.375591, -1.260323, -2.642154, -0.809912, 1.570796, 1.946387],accel_mss,speed_ms,0,blend_radius_m)
    |   movel([0.373465, -1.261222, -2.641661, -0.809506, 1.570796, 1.944261],accel_mss,speed_ms,0,blend_radius_m)
    |   movel([0.371679, -1.262240, -2.641102, -0.809047, 1.570796, 1.942475],accel_mss,speed_ms,0,blend_radius_m)
    |   movel([0.370221, -1.263354, -2.640488, -0.808547, 1.570796, 1.941017],accel_mss,speed_ms,0,blend_radius_m)
    |   movel([0.369081, -1.264541, -2.639833, -0.808015, 1.570796, 1.939877],accel_mss,speed_ms,0,blend_radius_m)
    |   movel([0.368250, -1.265773, -2.639151, -0.807465, 1.570796, 1.939047],accel_mss,speed_ms,0,blend_radius_m)
    |   movel([0.367715, -1.267031, -2.638453, -0.806905, 1.570796, 1.938511],accel_mss,speed_ms,0,blend_radius_m)
    |   movel([0.367461, -1.268294, -2.637750, -0.806345, 1.570796, 1.938257],accel_mss,speed_ms,0,blend_radius_m)
    |   movel([0.367753, -1.270740, -2.636382, -0.805266, 1.570796, 1.938550],accel_mss,speed_ms,0,blend_radius_m)
    |   movel([0.369028, -1.272943, -2.635145, -0.804301, 1.570796, 1.939824],accel_mss,speed_ms,0,blend_radius_m)
    |   movel([0.371192, -1.274732, -2.634135, -0.803522, 1.570796, 1.941988],accel_mss,speed_ms,0,blend_radius_m)
    |   movel([0.374149, -1.275949, -2.633446, -0.802994, 1.570796, 1.944945],accel_mss,speed_ms,0,blend_radius_m)
    |   movel([0.376221, -1.276261, -2.633270, -0.802859, 1.570796, 1.947017],accel_mss,speed_ms,0,blend_radius_m)
    |   movel([0.378885, -1.276306, -2.633244, -0.802839, 1.570796, 1.949681],accel_mss,speed_ms,0,blend_radius_m)
    |   movel([0.385680, -1.275714, -2.633579, -0.803095, 1.570796, 1.956477],accel_mss,speed_ms,0,blend_radius_m)
    |   movel([0.393907, -1.274431, -2.634305, -0.803653, 1.570796, 1.964703],accel_mss,speed_ms,0,blend_radius_m)
    |   movel([0.402941, -1.272692, -2.635286, -0.804411, 1.570796, 1.973738],accel_mss,speed_ms,0,blend_radius_m)
    |   movel([0.420926, -1.268739, -2.637502, -0.806149, 1.570796, 1.991723],accel_mss,speed_ms,0,blend_radius_m)
    |   movel([0.434579, -1.265470, -2.639319, -0.807600, 1.570796, 2.005375],accel_mss,speed_ms,0,blend_radius_m)
    |   movel([0.441461, -1.263813, -2.640235, -0.808341, 1.570796, 2.012257],accel_mss,speed_ms,0,blend_radius_m)
    |   movel([0.445192, -1.262796, -2.640796, -0.808797, 1.570796, 2.015988],accel_mss,speed_ms,0,blend_radius_m)
    |   movel([0.448060, -1.261769, -2.641361, -0.809259, 1.570796, 2.018856],accel_mss,speed_ms,0,blend_radius_m)
    |   movel([0.448856, -1.261320, -2.641607, -0.809461, 1.570796, 2.019653],accel_mss,speed_ms,0,blend_radius_m)
    |   movel([0.449190, -1.260915, -2.641830, -0.809644, 1.570796, 2.019986],accel_mss,speed_ms,0,blend_radius_m)
    |   movel([0.448849, -1.260012, -2.642325, -0.810053, 1.570796, 2.019645],accel_mss,speed_ms,0,blend_radius_m)
    |   movel([0.446786, -1.258184, -2.643323, -0.810882, 1.570796, 2.017582],accel_mss,speed_ms,0,blend_radius_m)
    |   movel([0.444119, -1.256850, -2.644049, -0.811490, 1.570796, 2.014916],accel_mss,speed_ms,0,blend_radius_m)
    |   movel([0.438114, -1.254328, -2.645416, -0.812645, 1.570796, 2.008910],accel_mss,speed_ms,0,blend_radius_m)
    |   movel([0.435336, -1.252464, -2.646421, -0.813504, 1.570796, 2.006132],accel_mss,speed_ms,0,blend_radius_m)
    |   movel([0.433086, -1.249732, -2.647887, -0.814770, 1.570796, 2.003882],accel_mss,speed_ms,0,blend_radius_m)
    |   movel([0.432250, -1.247928, -2.648850, -0.815611, 1.570796, 2.003046],accel_mss,speed_ms,0,blend_radius_m)
    |   movel([0.431650, -1.245772, -2.649996, -0.816621, 1.570796, 2.002446],accel_mss,speed_ms,0,blend_radius_m)
    |   movel([0.431326, -1.243215, -2.651348, -0.817826, 1.570796, 2.002123],accel_mss,speed_ms,0,blend_radius_m)
    |   movel([0.431319, -1.240207, -2.652928, -0.819254, 1.570796, 2.002115],accel_mss,speed_ms,0,blend_radius_m)
    |   movel([0.431929, -1.235989, -2.655126, -0.821273, 1.570796, 2.002725],accel_mss,speed_ms,0,blend_radius_m)
    |   movel([0.433276, -1.231767, -2.657306, -0.823316, 1.570796, 2.004073],accel_mss,speed_ms,0,blend_radius_m)
    |   movel([0.435284, -1.227549, -2.659463, -0.825377, 1.570796, 2.006081],accel_mss,speed_ms,0,blend_radius_m)
    |   movel([0.437866, -1.223356, -2.661587, -0.827446, 1.570796, 2.008662],accel_mss,speed_ms,0,blend_radius_m)
    |   movel([0.440932, -1.219202, -2.663671, -0.829516, 1.570796, 2.011728],accel_mss,speed_ms,0,blend_radius_m)
    |   movel([0.444393, -1.215110, -2.665705, -0.831574, 1.570796, 2.015189],accel_mss,speed_ms,0,blend_radius_m)
    |   movel([0.448159, -1.211095, -2.667682, -0.833612, 1.570796, 2.018955],accel_mss,speed_ms,0,blend_radius_m)
    |   movel([0.452132, -1.207183, -2.669591, -0.835615, 1.570796, 2.022928],accel_mss,speed_ms,0,blend_radius_m)
    |   movel([0.459963, -1.200287, -2.672915, -0.839186, 1.570796, 2.030760],accel_mss,speed_ms,0,blend_radius_m)
    |   movel([0.467141, -1.194888, -2.675481, -0.842019, 1.570796, 2.037937],accel_mss,speed_ms,0,blend_radius_m)
    |   movel([0.473315, -1.190913, -2.677350, -0.844126, 1.570796, 2.044112],accel_mss,speed_ms,0,blend_radius_m)
    |   movel([0.478143, -1.188273, -2.678582, -0.845534, 1.570796, 2.048939],accel_mss,speed_ms,0,blend_radius_m)
    |   movel([0.485280, -1.185195, -2.680009, -0.847185, 1.570796, 2.056076],accel_mss,speed_ms,0,blend_radius_m)
    |   movel([0.492132, -1.183154, -2.680950, -0.848286, 1.570796, 2.062928],accel_mss,speed_ms,0,blend_radius_m)
    |   movel([0.498614, -1.182134, -2.681418, -0.848837, 1.570796, 2.069410],accel_mss,speed_ms,0,blend_radius_m)
    |   movel([0.504640, -1.182106, -2.681431, -0.848852, 1.570796, 2.075437],accel_mss,speed_ms,0,blend_radius_m)
    |   movel([0.510130, -1.183037, -2.681003, -0.848349, 1.570796, 2.080927],accel_mss,speed_ms,0,blend_radius_m)
    |   movel([0.515015, -1.184882, -2.680154, -0.847354, 1.570796, 2.085811],accel_mss,speed_ms,0,blend_radius_m)
    |   movel([0.519222, -1.187594, -2.678898, -0.845897, 1.570796, 2.090018],accel_mss,speed_ms,0,blend_radius_m)
    |   movel([0.522688, -1.191123, -2.677252, -0.844014, 1.570796, 2.093484],accel_mss,speed_ms,0,blend_radius_m)
    |   movel([0.525123, -1.194952, -2.675451, -0.841986, 1.570796, 2.095919],accel_mss,speed_ms,0,blend_radius_m)
    |   movel([0.527099, -1.199116, -2.673475, -0.839798, 1.570796, 2.097895],accel_mss,speed_ms,0,blend_radius_m)
    |   movel([0.528957, -1.203267, -2.671485, -0.837636, 1.570796, 2.099753],accel_mss,speed_ms,0,blend_radius_m)
    |   movel([0.531040, -1.207069, -2.669647, -0.835673, 1.570796, 2.101836],accel_mss,speed_ms,0,blend_radius_m)
    |   movel([0.533681, -1.210200, -2.668121, -0.834069, 1.570796, 2.104477],accel_mss,speed_ms,0,blend_radius_m)
    |   movel([0.535315, -1.211411, -2.667527, -0.833451, 1.570796, 2.106112],accel_mss,speed_ms,0,blend_radius_m)
    |   movel([0.537212, -1.212339, -2.667072, -0.832979, 1.570796, 2.108009],accel_mss,speed_ms,0,blend_radius_m)
    |   movel([0.539416, -1.212941, -2.666775, -0.832673, 1.570796, 2.110213],accel_mss,speed_ms,0,blend_radius_m)
    |   movel([0.541968, -1.213181, -2.666657, -0.832551, 1.570796, 2.112765],accel_mss,speed_ms,0,blend_radius_m)
    |   movel([0.544915, -1.213019, -2.666737, -0.832633, 1.570796, 2.115712],accel_mss,speed_ms,0,blend_radius_m)
    |   movel([0.548300, -1.212413, -2.667035, -0.832941, 1.570796, 2.119096],accel_mss,speed_ms,0,blend_radius_m)
    |   movel([0.551384, -1.211420, -2.667523, -0.833446, 1.570796, 2.122181],accel_mss,speed_ms,0,blend_radius_m)
    |   movel([0.554099, -1.210012, -2.668212, -0.834164, 1.570796, 2.124896],accel_mss,speed_ms,0,blend_radius_m)
    |   movel([0.556436, -1.208270, -2.669063, -0.835057, 1.570796, 2.127233],accel_mss,speed_ms,0,blend_radius_m)
    |   movel([0.558399, -1.206275, -2.670032, -0.836082, 1.570796, 2.129195],accel_mss,speed_ms,0,blend_radius_m)
    |   movel([0.559977, -1.204108, -2.671080, -0.837201, 1.570796, 2.130773],accel_mss,speed_ms,0,blend_radius_m)
    |   movel([0.561161, -1.201857, -2.672163, -0.838369, 1.570796, 2.131957],accel_mss,speed_ms,0,blend_radius_m)
    |   movel([0.561946, -1.199608, -2.673240, -0.839541, 1.570796, 2.132742],accel_mss,speed_ms,0,blend_radius_m)
    |   movel([0.562323, -1.197448, -2.674269, -0.840672, 1.570796, 2.133120],accel_mss,speed_ms,0,blend_radius_m)
    |   movel([0.562282, -1.195470, -2.675206, -0.841712, 1.570796, 2.133079],accel_mss,speed_ms,0,blend_radius_m)
    |   movel([0.561814, -1.193766, -2.676011, -0.842612, 1.570796, 2.132610],accel_mss,speed_ms,0,blend_radius_m)
    |   movel([0.560908, -1.192428, -2.676640, -0.843321, 1.570796, 2.131704],accel_mss,speed_ms,0,blend_radius_m)
    |   movel([0.559557, -1.191549, -2.677052, -0.843787, 1.570796, 2.130353],accel_mss,speed_ms,0,blend_radius_m)
    |   movel([0.557757, -1.191217, -2.677208, -0.843964, 1.570796, 2.128553],accel_mss,speed_ms,0,blend_radius_m)
    |   movel([0.555502, -1.191529, -2.677062, -0.843798, 1.570796, 2.126299],accel_mss,speed_ms,0,blend_radius_m)
    |   movel([0.552789, -1.192575, -2.676571, -0.843243, 1.570796, 2.123586],accel_mss,speed_ms,0,blend_radius_m)
    |   movel([0.549621, -1.194433, -2.675696, -0.842260, 1.570796, 2.120417],accel_mss,speed_ms,0,blend_radius_m)
    |   movel([0.551314, -1.194767, -2.675539, -0.842083, 1.570796, 2.122110],accel_mss,speed_ms,0,blend_radius_m)
    |   movel([0.552501, -1.195444, -2.675219, -0.841726, 1.570796, 2.123297],accel_mss,speed_ms,0,blend_radius_m)
    |   movel([0.553173, -1.196410, -2.674761, -0.841218, 1.570796, 2.123969],accel_mss,speed_ms,0,blend_radius_m)
    |   movel([0.553328, -1.197614, -2.674190, -0.840585, 1.570796, 2.124125],accel_mss,speed_ms,0,blend_radius_m)
    |   movel([0.552957, -1.199009, -2.673526, -0.839854, 1.570796, 2.123754],accel_mss,speed_ms,0,blend_radius_m)
    |   movel([0.552057, -1.200542, -2.672793, -0.839054, 1.570796, 2.122853],accel_mss,speed_ms,0,blend_radius_m)
    |   movel([0.550623, -1.202161, -2.672017, -0.838211, 1.570796, 2.121419],accel_mss,speed_ms,0,blend_radius_m)
    |   movel([0.548649, -1.203819, -2.671219, -0.837350, 1.570796, 2.119445],accel_mss,speed_ms,0,blend_radius_m)
    |   movel([0.545042, -1.206062, -2.670135, -0.836192, 1.570796, 2.115838],accel_mss,speed_ms,0,blend_radius_m)
    |   movel([0.541785, -1.207268, -2.669550, -0.835571, 1.570796, 2.112581],accel_mss,speed_ms,0,blend_radius_m)
    |   movel([0.538887, -1.207544, -2.669416, -0.835429, 1.570796, 2.109683],accel_mss,speed_ms,0,blend_radius_m)
    |   movel([0.536375, -1.206992, -2.669684, -0.835713, 1.570796, 2.107171],accel_mss,speed_ms,0,blend_radius_m)
    |   movel([0.534273, -1.205702, -2.670310, -0.836377, 1.570796, 2.105069],accel_mss,speed_ms,0,blend_radius_m)
    |   movel([0.532608, -1.203767, -2.671244, -0.837377, 1.570796, 2.103405],accel_mss,speed_ms,0,blend_radius_m)
    |   movel([0.531417, -1.201279, -2.672440, -0.838669, 1.570796, 2.102213],accel_mss,speed_ms,0,blend_radius_m)
    |   movel([0.530724, -1.198329, -2.673850, -0.840210, 1.570796, 2.101521],accel_mss,speed_ms,0,blend_radius_m)
    |   movel([0.530576, -1.194998, -2.675429, -0.841961, 1.570796, 2.101372],accel_mss,speed_ms,0,blend_radius_m)
    |   movel([0.530999, -1.191386, -2.677129, -0.843874, 1.570796, 2.101795],accel_mss,speed_ms,0,blend_radius_m)
    |   movel([0.532040, -1.187576, -2.678906, -0.845907, 1.570796, 2.102836],accel_mss,speed_ms,0,blend_radius_m)
    |   movel([0.533730, -1.183673, -2.680711, -0.848005, 1.570796, 2.104527],accel_mss,speed_ms,0,blend_radius_m)
    |   movel([0.536115, -1.179766, -2.682501, -0.850122, 1.570796, 2.106911],accel_mss,speed_ms,0,blend_radius_m)
    |   movel([0.539226, -1.175962, -2.684228, -0.852199, 1.570796, 2.110022],accel_mss,speed_ms,0,blend_radius_m)
    |   movel([0.543102, -1.172367, -2.685846, -0.854175, 1.570796, 2.113898],accel_mss,speed_ms,0,blend_radius_m)
    |   movel([0.547771, -1.169094, -2.687308, -0.855987, 1.570796, 2.118568],accel_mss,speed_ms,0,blend_radius_m)
    |   movel([0.551250, -1.167142, -2.688175, -0.857072, 1.570796, 2.122046],accel_mss,speed_ms,0,blend_radius_m)
    |   movel([0.554711, -1.165505, -2.688898, -0.857986, 1.570796, 2.125507],accel_mss,speed_ms,0,blend_radius_m)
    |   movel([0.558121, -1.164182, -2.689481, -0.858726, 1.570796, 2.128917],accel_mss,speed_ms,0,blend_radius_m)
    |   movel([0.561453, -1.163189, -2.689917, -0.859283, 1.570796, 2.132250],accel_mss,speed_ms,0,blend_radius_m)
    |   movel([0.564675, -1.162525, -2.690208, -0.859655, 1.570796, 2.135471],accel_mss,speed_ms,0,blend_radius_m)
    |   movel([0.567760, -1.162198, -2.690352, -0.859839, 1.570796, 2.138557],accel_mss,speed_ms,0,blend_radius_m)
    |   movel([0.570678, -1.162213, -2.690345, -0.859831, 1.570796, 2.141474],accel_mss,speed_ms,0,blend_radius_m)
    |   movel([0.573401, -1.162569, -2.690189, -0.859631, 1.570796, 2.144197],accel_mss,speed_ms,0,blend_radius_m)
    |   movel([0.575897, -1.163272, -2.689881, -0.859236, 1.570796, 2.146694],accel_mss,speed_ms,0,blend_radius_m)
    |   movel([0.578144, -1.164319, -2.689421, -0.858649, 1.570796, 2.148941],accel_mss,speed_ms,0,blend_radius_m)
    |   movel([0.580112, -1.165714, -2.688806, -0.857869, 1.570796, 2.150908],accel_mss,speed_ms,0,blend_radius_m)
    |   movel([0.581777, -1.167457, -2.688035, -0.856897, 1.570796, 2.152573],accel_mss,speed_ms,0,blend_radius_m)
    |   movel([0.583111, -1.169543, -2.687108, -0.855738, 1.570796, 2.153907],accel_mss,speed_ms,0,blend_radius_m)
    |   movel([0.584095, -1.171969, -2.686025, -0.854395, 1.570796, 2.154891],accel_mss,speed_ms,0,blend_radius_m)
    |   movel([0.584699, -1.174738, -2.684781, -0.852871, 1.570796, 2.155496],accel_mss,speed_ms,0,blend_radius_m)
    |   movel([0.584905, -1.177843, -2.683376, -0.851170, 1.570796, 2.155702],accel_mss,speed_ms,0,blend_radius_m)
    |   movel([0.584309, -1.181285, -2.681807, -0.849297, 1.570796, 2.155106],accel_mss,speed_ms,0,blend_radius_m)
    |   movel([0.583006, -1.185212, -2.680001, -0.847176, 1.570796, 2.153802],accel_mss,speed_ms,0,blend_radius_m)
    |   movel([0.581714, -1.188620, -2.678421, -0.845348, 1.570796, 2.152510],accel_mss,speed_ms,0,blend_radius_m)
    |   movel([0.581138, -1.190527, -2.677531, -0.844331, 1.570796, 2.151935],accel_mss,speed_ms,0,blend_radius_m)
    |   movel([0.581828, -1.191469, -2.677090, -0.843830, 1.570796, 2.152624],accel_mss,speed_ms,0,blend_radius_m)
    |   movel([0.583400, -1.192577, -2.676570, -0.843242, 1.570796, 2.154196],accel_mss,speed_ms,0,blend_radius_m)
    |   movel([0.585132, -1.193800, -2.675995, -0.842594, 1.570796, 2.155928],accel_mss,speed_ms,0,blend_radius_m)
    |   movel([0.586312, -1.195070, -2.675396, -0.841924, 1.570796, 2.157108],accel_mss,speed_ms,0,blend_radius_m)
    |   movel([0.587182, -1.197307, -2.674336, -0.840746, 1.570796, 2.157979],accel_mss,speed_ms,0,blend_radius_m)
    |   movel([0.587557, -1.199696, -2.673198, -0.839495, 1.570796, 2.158354],accel_mss,speed_ms,0,blend_radius_m)
    |   movel([0.587471, -1.202201, -2.671998, -0.838190, 1.570796, 2.158267],accel_mss,speed_ms,0,blend_radius_m)
    |   movel([0.586960, -1.204781, -2.670755, -0.836853, 1.570796, 2.157757],accel_mss,speed_ms,0,blend_radius_m)
    |   movel([0.586065, -1.207402, -2.669485, -0.835502, 1.570796, 2.156861],accel_mss,speed_ms,0,blend_radius_m)
    |   movel([0.584821, -1.210023, -2.668207, -0.834159, 1.570796, 2.155617],accel_mss,speed_ms,0,blend_radius_m)
    |   movel([0.583264, -1.212614, -2.666936, -0.832839, 1.570796, 2.154060],accel_mss,speed_ms,0,blend_radius_m)
    |   movel([0.581429, -1.215136, -2.665692, -0.831561, 1.570796, 2.152225],accel_mss,speed_ms,0,blend_radius_m)
    |   movel([0.579347, -1.217560, -2.664489, -0.830339, 1.570796, 2.150144],accel_mss,speed_ms,0,blend_radius_m)
    |   movel([0.577056, -1.219850, -2.663347, -0.829192, 1.570796, 2.147852],accel_mss,speed_ms,0,blend_radius_m)
    |   movel([0.574585, -1.221975, -2.662282, -0.828132, 1.570796, 2.145381],accel_mss,speed_ms,0,blend_radius_m)
    |   speed_ms = 0.003
    |   movel([0.574585, -1.214836, -2.658735, -0.838818, 1.570796, 2.145381],accel_mss,speed_ms,0,blend_radius_m)
    |   speed_ms = 0.05
    |   movel([0.574585, -1.187672, -2.644287, -0.880430, 1.570796, 2.145381],accel_mss,speed_ms,0,blend_radius_m)
    |   #M_RunCode9
    |   movel([0.591130, -1.186616, -2.644793, -0.880980, 1.570796, 2.161926],accel_mss,speed_ms,0,blend_radius_m)
    |   #M_RunCode3
    |   movel([0.591130, -1.213790, -2.659255, -0.839344, 1.570796, 2.161926],accel_mss,speed_ms,0,blend_radius_m)
    |   speed_ms = 0.003
    |   movel([0.591130, -1.220931, -2.662806, -0.828652, 1.570796, 2.161926],accel_mss,speed_ms,0,blend_radius_m)
    |   speed_ms = 0.02
    |   movel([0.592137, -1.218745, -2.663899, -0.829745, 1.570796, 2.162934],accel_mss,speed_ms,0,blend_radius_m)
    |   movel([0.594754, -1.214294, -2.666108, -0.831987, 1.570796, 2.165550],accel_mss,speed_ms,0,blend_radius_m)
    |   movel([0.597117, -1.209933, -2.668251, -0.834205, 1.570796, 2.167913],accel_mss,speed_ms,0,blend_radius_m)
    |   movel([0.597804, -1.207861, -2.669262, -0.835266, 1.570796, 2.168601],accel_mss,speed_ms,0,blend_radius_m)
    |   movel([0.597944, -1.205900, -2.670214, -0.836275, 1.570796, 2.168741],accel_mss,speed_ms,0,blend_radius_m)
    |   movel([0.598344, -1.207080, -2.669642, -0.835668, 1.570796, 2.169140],accel_mss,speed_ms,0,blend_radius_m)
    |   movel([0.598528, -1.209517, -2.668454, -0.834418, 1.570796, 2.169324],accel_mss,speed_ms,0,blend_radius_m)
    |   movel([0.598052, -1.212011, -2.667233, -0.833146, 1.570796, 2.168849],accel_mss,speed_ms,0,blend_radius_m)
    |   movel([0.597124, -1.214544, -2.665985, -0.831860, 1.570796, 2.167920],accel_mss,speed_ms,0,blend_radius_m)
    |   movel([0.595945, -1.217100, -2.664718, -0.830571, 1.570796, 2.166742],accel_mss,speed_ms,0,blend_radius_m)
    |   movel([0.593649, -1.222221, -2.662158, -0.828010, 1.570796, 2.164445],accel_mss,speed_ms,0,blend_radius_m)
    |   movel([0.592927, -1.224757, -2.660879, -0.826753, 1.570796, 2.163723],accel_mss,speed_ms,0,blend_radius_m)
    |   movel([0.592753, -1.227254, -2.659613, -0.825522, 1.570796, 2.163549],accel_mss,speed_ms,0,blend_radius_m)
    |   movel([0.593152, -1.229808, -2.658310, -0.824271, 1.570796, 2.163949],accel_mss,speed_ms,0,blend_radius_m)
    |   movel([0.593515, -1.231090, -2.657654, -0.823646, 1.570796, 2.164311],accel_mss,speed_ms,0,blend_radius_m)
    |   movel([0.593934, -1.231695, -2.657343, -0.823351, 1.570796, 2.164730],accel_mss,speed_ms,0,blend_radius_m)
    |   movel([0.595385, -1.231170, -2.657612, -0.823606, 1.570796, 2.166182],accel_mss,speed_ms,0,blend_radius_m)
    |   movel([0.596567, -1.230799, -2.657803, -0.823787, 1.570796, 2.167363],accel_mss,speed_ms,0,blend_radius_m)
    |   movel([0.597729, -1.230654, -2.657877, -0.823858, 1.570796, 2.168526],accel_mss,speed_ms,0,blend_radius_m)
    |   movel([0.599793, -1.230918, -2.657742, -0.823729, 1.570796, 2.170590],accel_mss,speed_ms,0,blend_radius_m)
    |   movel([0.601137, -1.231489, -2.657449, -0.823451, 1.570796, 2.171934],accel_mss,speed_ms,0,blend_radius_m)
    |   movel([0.601916, -1.232321, -2.657021, -0.823047, 1.570796, 2.172712],accel_mss,speed_ms,0,blend_radius_m)
    |   movel([0.602283, -1.233378, -2.656477, -0.822534, 1.570796, 2.173080],accel_mss,speed_ms,0,blend_radius_m)
    |   movel([0.602404, -1.236006, -2.655118, -0.821265, 1.570796, 2.173201],accel_mss,speed_ms,0,blend_radius_m)
    |   movel([0.602732, -1.239072, -2.653522, -0.819795, 1.570796, 2.173529],accel_mss,speed_ms,0,blend_radius_m)
    |   movel([0.603956, -1.242758, -2.651589, -0.818043, 1.570796, 2.174752],accel_mss,speed_ms,0,blend_radius_m)
    |   movel([0.605339, -1.246307, -2.649712, -0.816370, 1.570796, 2.176135],accel_mss,speed_ms,0,blend_radius_m)
    |   movel([0.606495, -1.249975, -2.647757, -0.814657, 1.570796, 2.177291],accel_mss,speed_ms,0,blend_radius_m)
    |   movel([0.607055, -1.253999, -2.645593, -0.812796, 1.570796, 2.177851],accel_mss,speed_ms,0,blend_radius_m)
    |   movel([0.606957, -1.256363, -2.644313, -0.811712, 1.570796, 2.177754],accel_mss,speed_ms,0,blend_radius_m)
    |   movel([0.606574, -1.258814, -2.642979, -0.810596, 1.570796, 2.177370],accel_mss,speed_ms,0,blend_radius_m)
    |   movel([0.605240, -1.263850, -2.640215, -0.808324, 1.570796, 2.176037],accel_mss,speed_ms,0,blend_radius_m)
    |   movel([0.603630, -1.268869, -2.637429, -0.806091, 1.570796, 2.174427],accel_mss,speed_ms,0,blend_radius_m)
    |   movel([0.602317, -1.273627, -2.634759, -0.804002, 1.570796, 2.173113],accel_mss,speed_ms,0,blend_radius_m)
    |   movel([0.601117, -1.281213, -2.630445, -0.800731, 1.570796, 2.171914],accel_mss,speed_ms,0,blend_radius_m)
    |   movel([0.600699, -1.284417, -2.628601, -0.799371, 1.570796, 2.171495],accel_mss,speed_ms,0,blend_radius_m)
    |   movel([0.600093, -1.287488, -2.626821, -0.798080, 1.570796, 2.170889],accel_mss,speed_ms,0,blend_radius_m)
    |   movel([0.599084, -1.290613, -2.624998, -0.796778, 1.570796, 2.169881],accel_mss,speed_ms,0,blend_radius_m)
    |   movel([0.597449, -1.293977, -2.623022, -0.795390, 1.570796, 2.168245],accel_mss,speed_ms,0,blend_radius_m)
    |   movel([0.594970, -1.297762, -2.620781, -0.793846, 1.570796, 2.165767],accel_mss,speed_ms,0,blend_radius_m)
    |   movel([0.591443, -1.302146, -2.618162, -0.792081, 1.570796, 2.162240],accel_mss,speed_ms,0,blend_radius_m)
    |   movel([0.588290, -1.305535, -2.616120, -0.790733, 1.570796, 2.159086],accel_mss,speed_ms,0,blend_radius_m)
    |   movel([0.585156, -1.308447, -2.614354, -0.789587, 1.570796, 2.155953],accel_mss,speed_ms,0,blend_radius_m)
    |   movel([0.582045, -1.310910, -2.612852, -0.788627, 1.570796, 2.152841],accel_mss,speed_ms,0,blend_radius_m)
    |   movel([0.578950, -1.312954, -2.611599, -0.787836, 1.570796, 2.149747],accel_mss,speed_ms,0,blend_radius_m)
    |   movel([0.575884, -1.314607, -2.610582, -0.787200, 1.570796, 2.146680],accel_mss,speed_ms,0,blend_radius_m)
    |   movel([0.572842, -1.315895, -2.609787, -0.786707, 1.570796, 2.143638],accel_mss,speed_ms,0,blend_radius_m)
    |   movel([0.569832, -1.316841, -2.609202, -0.786346, 1.570796, 2.140628],accel_mss,speed_ms,0,blend_radius_m)
    |   movel([0.566853, -1.317471, -2.608811, -0.786107, 1.570796, 2.137650],accel_mss,speed_ms,0,blend_radius_m)
    |   movel([0.563917, -1.317807, -2.608603, -0.785979, 1.570796, 2.134713],accel_mss,speed_ms,0,blend_radius_m)
    |   movel([0.561020, -1.317874, -2.608561, -0.785954, 1.570796, 2.131816],accel_mss,speed_ms,0,blend_radius_m)
    |   movel([0.555372, -1.317283, -2.608928, -0.786178, 1.570796, 2.126169],accel_mss,speed_ms,0,blend_radius_m)
    |   movel([0.549959, -1.315871, -2.609802, -0.786716, 1.570796, 2.120755],accel_mss,speed_ms,0,blend_radius_m)
    |   movel([0.544828, -1.313808, -2.611074, -0.787507, 1.570796, 2.115624],accel_mss,speed_ms,0,blend_radius_m)
    |   movel([0.540380, -1.311340, -2.612589, -0.788460, 1.570796, 2.111176],accel_mss,speed_ms,0,blend_radius_m)
    |   movel([0.534758, -1.308061, -2.614590, -0.789739, 1.570796, 2.105554],accel_mss,speed_ms,0,blend_radius_m)
    |   movel([0.528188, -1.304821, -2.616552, -0.791016, 1.570796, 2.098984],accel_mss,speed_ms,0,blend_radius_m)
    |   movel([0.524628, -1.303480, -2.617360, -0.791549, 1.570796, 2.095425],accel_mss,speed_ms,0,blend_radius_m)
    |   movel([0.520928, -1.302465, -2.617971, -0.791953, 1.570796, 2.091724],accel_mss,speed_ms,0,blend_radius_m)
    |   movel([0.517131, -1.301883, -2.618320, -0.792186, 1.570796, 2.087927],accel_mss,speed_ms,0,blend_radius_m)
    |   movel([0.513273, -1.301833, -2.618350, -0.792206, 1.570796, 2.084070],accel_mss,speed_ms,0,blend_radius_m)
    |   movel([0.509398, -1.302418, -2.617999, -0.791972, 1.570796, 2.080194],accel_mss,speed_ms,0,blend_radius_m)
    |   movel([0.505555, -1.303731, -2.617209, -0.791449, 1.570796, 2.076351],accel_mss,speed_ms,0,blend_radius_m)
    |   movel([0.503656, -1.304691, -2.616630, -0.791068, 1.570796, 2.074453],accel_mss,speed_ms,0,blend_radius_m)
    |   movel([0.501784, -1.305870, -2.615918, -0.790601, 1.570796, 2.072580],accel_mss,speed_ms,0,blend_radius_m)
    |   movel([0.499943, -1.307273, -2.615068, -0.790048, 1.570796, 2.070740],accel_mss,speed_ms,0,blend_radius_m)
    |   movel([0.498139, -1.308914, -2.614070, -0.789405, 1.570796, 2.068936],accel_mss,speed_ms,0,blend_radius_m)
    |   movel([0.496379, -1.310806, -2.612916, -0.788667, 1.570796, 2.067175],accel_mss,speed_ms,0,blend_radius_m)
    |   movel([0.494666, -1.312954, -2.611599, -0.787835, 1.570796, 2.065462],accel_mss,speed_ms,0,blend_radius_m)
    |   movel([0.491414, -1.318062, -2.608445, -0.785883, 1.570796, 2.062211],accel_mss,speed_ms,0,blend_radius_m)
    |   movel([0.490466, -1.320566, -2.606885, -0.784938, 1.570796, 2.061262],accel_mss,speed_ms,0,blend_radius_m)
    |   movel([0.489985, -1.323060, -2.605324, -0.784005, 1.570796, 2.060781],accel_mss,speed_ms,0,blend_radius_m)
